MAIN.stLine_BH0IPL.fbLine(stLine:=MAIN.stLine_BH0IPL);
MAIN.stLine_BH0IPL.stStation_BH0IPL01.fbStation(
				stLine:=MAIN.stLine_BH0IPL,
				stStation:=MAIN.stLine_BH0IPL.stStation_BH0IPL01);

END_PROGRAM

// ---- POUs/Program_PIM_Lines/HP/BH0JPL_LineBackground.TcPOU
PROGRAM BH0JPL_LineBackground
VAR
END_VAR

MAIN.stLine_BH0JPL.fbLine(stLine:=MAIN.stLine_BH0JPL);
MAIN.stLine_BH0JPL.stStation_BH0JPL01.fbStation(
				stLine:=MAIN.stLine_BH0JPL,
				stStation:=MAIN.stLine_BH0JPL.stStation_BH0JPL01);

END_PROGRAM

// ---- POUs/Program_PIM_Lines/HP/BH0KPL_LineBackground.TcPOU
PROGRAM BH0KPL_LineBackground
VAR
END_VAR

MAIN.stLine_BH0KPL.fbLine(stLine:=MAIN.stLine_BH0KPL);
MAIN.stLine_BH0KPL.stStation_BH0KPL01.fbStation(
				stLine:=MAIN.stLine_BH0KPL,
				stStation:=MAIN.stLine_BH0KPL.stStation_BH0KPL01);

END_PROGRAM

// ---- POUs/Program_PIM_Lines/HP/BH0LPL_LineBackground.TcPOU
PROGRAM BH0LPL_LineBackground
VAR
END_VAR

MAIN.stLine_BH0LPL.fbLine(stLine:=MAIN.stLine_BH0LPL);
MAIN.stLine_BH0LPL.stStation_BH0LPL01.fbStation(
				stLine:=MAIN.stLine_BH0LPL,
				stStation:=MAIN.stLine_BH0LPL.stStation_BH0LPL01);

END_PROGRAM

// ---- POUs/Program_PIM_Lines/HP/BH0MPL_LineBackground.TcPOU
PROGRAM BH0MPL_LineBackground
VAR
END_VAR

MAIN.stLine_BH0MPL.fbLine(stLine:=MAIN.stLine_BH0MPL);
MAIN.stLine_BH0MPL.stStation_BH0MPL01.fbStation(
				stLine:=MAIN.stLine_BH0MPL,
				stStation:=MAIN.stLine_BH0MPL.stStation_BH0MPL01);

END_PROGRAM

// ---- POUs/Checks/CheckBounds.TcPOU
// Implicitly generated code : DO NOT EDIT
FUNCTION CheckBounds : DINT
VAR_INPUT
	index, lower, upper: DINT;
END_VAR

// Implicitly generated code : Only an Implementation suggestion
{noflow}
IF  index < lower THEN
	GVL_Checks.diCheckBounds := GVL_Checks.diCheckBounds +1;
	CheckBounds := lower;
ELSIF  index > upper THEN
	GVL_Checks.diCheckBounds := GVL_Checks.diCheckBounds +1;
	CheckBounds := upper;
ELSE  
	CheckBounds := index;
END_IF
{flow}

END_FUNCTION

// ---- POUs/Checks/CheckDivDInt.TcPOU
// Implicitly generated code : DO NOT EDIT
FUNCTION CheckDivDInt : DINT
VAR_INPUT
	divisor:DINT;
END_VAR

// Implicitly generated code : Only an Implementation suggestion
{noflow}
IF divisor = 0 THEN
	GVL_Checks.diCheckDivDInt := GVL_Checks.diCheckDivDInt +1;
	CheckDivDInt:=1;
ELSE
	CheckDivDInt:=divisor;
END_IF;
{flow}

END_FUNCTION

// ---- POUs/Checks/CheckDivLInt.TcPOU
// Implicitly generated code : DO NOT EDIT
FUNCTION CheckDivLInt : LINT
VAR_INPUT
	divisor:LINT;
END_VAR

// Implicitly generated code : Only an Implementation suggestion
{noflow}
IF divisor = 0 THEN
GVL_Checks.diCheckDivLInt := GVL_Checks.diCheckDivLInt +1;
	CheckDivLInt:=1;
ELSE
	CheckDivLInt:=divisor;
END_IF;
{flow}

END_FUNCTION

// ---- POUs/Checks/CheckDivLReal.TcPOU
// Implicitly generated code : DO NOT EDIT
FUNCTION CheckDivLReal : LREAL
VAR_INPUT
	divisor:LREAL;
END_VAR

// Implicitly generated code : Only an Implementation suggestion
{noflow}
IF divisor = 0 THEN
	GVL_Checks.diCheckDivLReal := GVL_Checks.diCheckDivLReal +1;
	CheckDivLReal:=1;
ELSE
	CheckDivLReal:=divisor;
END_IF;
{flow}

END_FUNCTION

// ---- POUs/Checks/CheckDivReal.TcPOU
// Implicitly generated code : DO NOT EDIT
FUNCTION CheckDivReal : REAL
VAR_INPUT
	divisor:REAL;
END_VAR

// Implicitly generated code : Only an Implementation suggestion
{noflow}
IF divisor = 0 THEN
GVL_Checks.diCheckDivReal := GVL_Checks.diCheckDivReal +1;
	CheckDivReal:=1;
ELSE
	CheckDivReal:=divisor;
END_IF;
{flow}

END_FUNCTION

// ---- POUs/Checks/CheckLRangeSigned.TcPOU
// Implicitly generated code : DO NOT EDIT
FUNCTION CheckLRangeSigned : LINT
VAR_INPUT
	value, lower, upper: LINT;
END_VAR

// Implicitly generated code : Only an Implementation suggestion
{noflow}
IF (value < lower) THEN
	GVL_Checks.diCheckLRangeSigned := GVL_Checks.diCheckLRangeSigned +1;
	CheckLRangeSigned := lower;
ELSIF(value > upper) THEN
	GVL_Checks.diCheckLRangeSigned := GVL_Checks.diCheckLRangeSigned +1;
	CheckLRangeSigned := upper;
ELSE
	CheckLRangeSigned := value;
END_IF

{flow}

END_FUNCTION

// ---- POUs/Checks/CheckLRangeUnsigned.TcPOU
// Implicitly generated code : DO NOT EDIT
FUNCTION CheckLRangeUnsigned : ULINT
VAR_INPUT
	value, lower, upper: ULINT;
END_VAR

// Implicitly generated code : Only an Implementation suggestion
{noflow}
IF (value < lower) THEN
	GVL_Checks.diCheckLRangeUnsigned := GVL_Checks.diCheckLRangeUnsigned +1;
	CheckLRangeUnsigned := lower;
ELSIF(value > upper) THEN
	GVL_Checks.diCheckLRangeUnsigned := GVL_Checks.diCheckLRangeUnsigned +1;
	CheckLRangeUnsigned := upper;
ELSE
	CheckLRangeUnsigned := value;
END_IF
{flow}

END_FUNCTION

// ---- POUs/Checks/CheckPointer.TcPOU
// Implicitly generated code : DO NOT EDIT
FUNCTION CheckPointer : POINTER TO BYTE
VAR_INPUT 
	ptToTest : POINTER TO BYTE; // Destination address of the pointer
	iSize : DINT;		        // Size of the type the pointer points to. (e.g: 20 for POINTER TO ARRAY [0..9] OF INT) 
	iGran : DINT;		        // Granularity of the pointer access. This is the size of the biggest non-structured data type in the type the pointer points to. (e.g: 2 for POINTER TO ARRAY [0..9] OF INT)
	bWrite: BOOL;		        // Indicates read or write Access. TRUE = write access.
END_VAR

// No standard way of implementation. Fill your own code here
CheckPointer := ptToTest;
IF ptToTest = 0 THEN
	GVL_Checks.diCheckPointer := GVL_Checks.diCheckPointer +1;	
END_IF
{flow}

END_FUNCTION

// ---- POUs/Checks/CheckRangeSigned.TcPOU
// Implicitly generated code : DO NOT EDIT
FUNCTION CheckRangeSigned : DINT
VAR_INPUT
	value, lower, upper: DINT;
END_VAR

// Implicitly generated code : Only an Implementation suggestion
{noflow}
IF (value < lower) THEN
	GVL_Checks.diCheckRangeSigned := GVL_Checks.diCheckRangeSigned +1;
	CheckRangeSigned := lower;
ELSIF(value > upper) THEN
	GVL_Checks.diCheckRangeSigned := GVL_Checks.diCheckRangeSigned +1;
	CheckRangeSigned := upper;
ELSE
	CheckRangeSigned := value;
END_IF
{flow}

END_FUNCTION

// ---- POUs/Checks/CheckRangeUnsigned.TcPOU
// Implicitly generated code : DO NOT EDIT
FUNCTION CheckRangeUnsigned : UDINT
VAR_INPUT
	value, lower, upper: UDINT;
END_VAR

// Implicitly generated code : Only an Implementation suggestion
{noflow}
IF (value < lower) THEN
	GVL_Checks.diCheckRangeUnsigned := GVL_Checks.diCheckRangeUnsigned +1;
	CheckRangeUnsigned := lower;
ELSIF(value > upper) THEN
	GVL_Checks.diCheckRangeUnsigned := GVL_Checks.diCheckRangeUnsigned +1;
	CheckRangeUnsigned := upper;
ELSE
	CheckRangeUnsigned := value;
END_IF
{flow}

END_FUNCTION

// ---- GlobalTextList.TcGTLO
TEXTLIST GlobalTextList
  2028 = '\tWelding plate heaters monitor settings'
  3970 = '\tWelding plate settings'
  1010 = '          Axis brake settings' | pl: 'Ustawienia hamulca'
  2001 = '          Manual mode'
  1107 = '       Actual process data'
  2145 = '       Aux settings'
  810 = '       Axis Calibration'
  1209 = '       Axis specific settings'
  1578 = '       General settings'
  2691 = '       PIM System Active' | pl: '      System PIM aktywny'
  2786 = '      Heat stamp'
  247 = '     %s'
  1851 = '     Heather checking'
  3653 = '    Assembly post station: %s' | pl: 'Stacja montażowa: %s'
  510 = '    Set packing station: %s' | pl: 'Stanowisko pakowania zest.: %s'
  842 = '%.0f'
  641 = '%.1f'
  852 = '%.1f [ % ]'
  5639 = '%.1f [ deg/s ]'
  714 = '%.1f [ mm/s ]'
  2700 = '%.1f [ N ]'
  543 = '%.1f [N]'
  382 = '%.1f [s]'
  978 = '%.2f'
  3732 = '%.2f [ deg ]'
  2622 = '%.2f [ mm ]'
  170 = '%.2f [deg]'
  1131 = '%.3f'
  2649 = '%.3f [ mm ]'
  283 = '%1.2f'
  8 = '%1.f'
  53 = '%2.2f'
  1254 = '%2.f'
  3164 = '%3.f'
  2235 = '%d'
  224 = '%d [deg/s2]'
  2693 = '%d [deg/s]'
  3397 = '%d [deg]'
  4376 = '%f'
  2797 = '%f.2'
  4602 = '%r'
  1 = '%s'
  3861 = "'"
  4535 = '+'
  897 = '+/- %2.2f'
  1682 = '-'
  2248 = '/\\ /\\ /\\      Set NEW    /\\ /\\ /\\' | pl: '/\\ /\\ /\\ Ustaw NOWE /\\ /\\ /\\' | gb: '/\\ /\\ /\\      Set NEW    /\\ /\\ /\\'
  1420 = '1. Adjustment (melting)'
  559 = '1. Choose\nCalibration'
  967 = '2. Connecting parts'
  1292 = '2. Prepare\npart templates'
  33 = '2a- Axis Up \nPart clamp'
  444 = '2b- Axis Dn \nPart clamp'
  2245 = '2c- Close\nWorkCover'
  347 = '3. Evaluate \nresults and exit calib.'
  2022 = '3a- Exit and\nsave result'
  1612 = '3b- Exit \nwithout save'
  393 = '< Act'
  700 = '<A'
  2014 = 'Aby dokonać resetu zaloguj się kartą'
  3442 = 'Aby dokonać resetu zaloguj się:\nswoją kartą'
  4965 = 'Aby dokonać resetu zaloguj się:\nswoją kartą, przykład: id_Pxxxx'
  522 = 'Aby dokonać resetu zaloguj się:\nswoją kartą, przykład: id_Pxxxx\nZalogowane konto ma \nwyświetlać imie i nazwisko'
  610 = 'Aby dokonać resetu zaloguj się:\nswoją kartą, przykład: id_Pxxxx\nZalogowane konto ma wyświetlać imie i nazwisko'
  3960 = 'Acceleration' | pl: 'Przyspieszenie'
  2097 = 'Act axis brake mode'
  2069 = 'Act val. [°C]'
  1347 = 'Activate/deactivate PIM' | pl: 'Włącz/Wyłącz PIM'
  1794 = 'Actual' | pl: 'Aktualne' | gb: 'Actual'
  308 = 'Actual Diference [%]'
  4954 = 'Actual error:' | pl: 'Obecny błąd:'
  1846 = 'Actual position' | pl: 'Obecna pozycja'
  2597 = 'Actual record'
  577 = 'Actual User: %s'
  1769 = 'Actual velocity' | pl: 'Obecna predkosc'
  4416 = 'Actual weight' | pl: 'Obecna waga'
  2569 = 'Actual weight offset [g]'
  1704 = 'Actual weight [g]' | pl: 'Obecna waga [g]'
  2451 = 'Actuator'
  3860 = 'Actuator state'
  685 = 'Adhesion force limit [ N]'
  1373 = 'Adjustment (melting) mode'
  4221 = 'Adjustment distance [mm]'
  2731 = 'Adjustment force [N]'
  743 = 'Adjustment timeout [s]'
  3068 = 'Admin' | pl: 'Administrator'
  1573 = 'Air cut valve acitive' | pl: 'Zawór odcinający powietrze'
  787 = 'Air supply active' | pl: 'Zasilanie pneumatyki włączone'
  1531 = 'Aktualna wartość położenia' | pl: 'Aktualna wartość położenia'
  360 = 'Alarm' | pl: 'Alarm'
  3603 = 'Alarm logging level settings' | pl: 'Poziom logowania alarmów'
  4801 = 'Amount of data exchange'
  4645 = 'Amount of errors'
  3292 = 'Amount of NG commands'
  3000 = 'Amount of OK commands'
  8057 = 'Auto Tare' | pl: 'Auto Tarowanie'
  1112 = 'Available recipe list:' | pl: 'Dostępne receptury:' | gb: 'Avaliable recipes:'
  39 = 'Axis DN WorkStep'
  1058 = 'Axis Down'
  1840 = 'Axis Down WorkStep:'
  561 = 'Axis power control'
  1525 = 'Axis UP WorkStep'
  1687 = 'Axis Up WorkStep:'
  915 = 'Axis Up:'
  195 = 'B02PL production line (LW)' | pl: 'Linia produkcyjna B02PL (LW)'
  1077 = 'BA02PL'
  3259 = 'BA02PL - 1'
  875 = 'BA02PL - 2'
  10432 = 'BA02PL.01.1'
  13845 = 'BA02PL.01.2'
  7111 = 'BA02PL.02'
  17460 = 'BA02PL.03'
  4811 = 'BA02PL.04'
  2952 = 'BA02PL.05'
  12157 = 'BA02PL.06.1'
  3189 = 'BA02PL.06.2'
  1729 = 'BA02PL01_M1'
  223 = 'BA02PL01_M1\nBA02PL01_M2\nBA02PL03'
  2992 = 'BA02PL01_M2'
  5907 = 'BA02PL02'
  2491 = 'BA02PL02\nBA02PL04'
  1317 = 'BA02PL03'
  4279 = 'BA02PL04'
  2606 = 'BA02PL05'
  4490 = 'BA02PL05 - SEQ'
  463 = 'BA02PL06_M1'
  89 = 'BA02PL06_M1\nBA02PL06_M2'
  5291 = 'BA02PL06_M2'
  2816 = 'BA02PL07'
  126 = 'Base pos'
  3252 = 'BB02PL'
  12665 = 'BB02PL.01'
  4132 = 'BB02PL01'
  4062 = 'BH0GPL'
  5405 = 'BH0GPL01_M1'
  4387 = 'BH0GPL01_M2'
  1088 = 'BH0GPL01_M3'
  1316 = 'BH0GPL_M1'
  1606 = 'BH0GPL_M2'
  3567 = 'BH0GPL_M3'
  2067 = 'BH0HPL'
  901 = 'BH0HPL01_M1'
  4474 = 'BH0HPL01_M2'
  1154 = 'BH0HPL01_M3'
  6321 = 'BH0IPL'
  5679 = 'BH0IPL01_M1'
  3354 = 'BH0IPL01_M2'
  197 = 'BH0IPL01_M3'
  6045 = 'BH0JPL'
  1356 = 'BH0JPL01_M1'
  1184 = 'BH0JPL01_M2'
  2515 = 'BH0JPL01_M3'
  3047 = 'BH0KPL'
  4183 = 'BH0KPL01_M1'
  2252 = 'BH0KPL01_M2'
  4613 = 'BH0KPL01_M3'
  778 = 'BH0LPL'
  1170 = 'BH0LPL01_M1'
  5197 = 'BH0LPL01_M2'
  4799 = 'BH0LPL01_M3'
  3559 = 'BH0MPL'
  350 = 'BH0MPL01_M1'
  4743 = 'BH0MPL01_M2'
  316 = 'BH0MPL01_M3'
  2507 = 'Block cardrige'
  3243 = 'Block perform'
  2953 = 'Blocker Down'
  3876 = 'Blocker Entrace'
  3364 = 'Blocker Escape'
  3696 = 'Blocker Input'
  573 = 'Blocker Output'
  3543 = 'Blocker Up'
  1981 = 'BO02PL'
  5711 = 'BO02PL.01'
  14356 = 'BO02PL.02'
  3039 = 'BO02PL01'
  5696 = 'BO02PL02'
  6799 = 'Bottle Detecion From %.2f' | pl: 'Wykrycie Butelki Od %.2f'
  2040 = 'Bottle Detecion To %.2f' | pl: 'Wykrycie Butelki Do %.2f'
  2283 = 'Bottle Incomming'
  3452 = 'Bottle Input'
  8074 = 'Bottle Separation' | pl: 'Oddzielanie Butelek'
  4027 = 'Box target weight: %.3f [kg]' | pl: 'Oczekiwana waga boxa: %.3f [kg]'
  5852 = 'BS02PL'
  8714 = 'BS02PL.01'
  5354 = 'BS02PL01'
  376 = 'BS02PL01_M1'
  701 = 'BS02PL01_M2'
  361 = 'BS02PL03'
  396 = 'BS02PL06_M1'
  649 = 'BS02PL06_M2'
  955 = 'Busy'
  3336 = 'Button On/Off'
  3328 = 'CA03PL'
  1865 = 'CA03PL11'
  2294 = 'CA03PL12'
  2710 = 'CA03PL13'
  514 = 'CA03PL14'
  2017 = 'CA03PL15'
  533 = 'CA03PL16'
  173 = 'CA03PL17'
  3355 = 'CA03PL18'
  200 = 'CA03PL19_M1'
  201 = 'CA03PL19_M2'
  1273 = 'CA03PL20'
  1845 = 'CA03PL21'
  3251 = 'CA03PL22'
  419 = 'Calibration'
  1260 = 'Calibration\nInProgress'
  303 = 'Calibration Target Data'
  179 = 'Camera Contrast'
  437 = 'Camera Exposure Time [us]'
  761 = 'Camera Gain Raw '
  248 = 'Camera Gamma'
  2217 = 'Camera Settings'
  516 = 'Cancel change' | pl: 'Anuluj zmiany' | gb: 'Cancel change'
  2722 = 'Cardrige Chamber'
  557 = 'Cardrige Input'
  90 = 'Cardrige Output'
  4204 = 'Cardrige Table'
  1549 = 'Chamber bussy'
  2795 = 'chamber cardrige'
  2343 = 'Chamber cardrige'
  3054 = 'Chamber work allow'
  7 = 'Check HeatedPlate heaters damage'
  1854 = 'Check heaters'
  109 = 'Check out part dimmenisons tolerance'
  1418 = 'Check part tolerance after contact'
  2132 = 'Check seal'
  5762 = 'Check Vision' | pl: 'Sprawdzanie Wizyjne'
  4753 = 'Check weight' | pl: 'Sprawdzanie wagi'
  5761 = 'Check Weight' | pl: 'Sprawdzanie Wagi'
  3524 = 'Ciśnienie szukania'
  1718 = 'Ciśnienie wprasowania'
  1684 = 'Clean errors' | pl: 'Wyczyść błędy'
  1086 = 'Clear\nStatistic'
  433 = 'Clear History'
  637 = 'CLOSE' | pl: 'ZAMKNIJ'
  1001 = 'Closed'
  508 = 'Closed \n(hiden)'
  654 = 'Closed (hiden)'
  812 = 'CM03PL'
  2300 = 'Cognex settings'
  519 = 'Colision detection EN'
  3451 = 'Colision force treshold'
  2838 = 'Communication Active'
  1552 = 'Communication Cycle Time'
  1968 = 'Communication Cycle Time [s]'
  908 = 'Communication Interval[s]'
  2124 = 'Communication IP'
  520 = 'Communication Ready'
  2647 = 'Confirm change !' | pl: 'Potwierdź zmiany'
  409 = 'Confirm error'
  4955 = 'Confirm PIM Alarm' | pl: 'Potwierdź alarm PIM'
  1985 = 'Confirm PLC Alarm' | pl: 'Potwierdź alarm PLC'
  883 = 'Conn. contact point detec. force [N]'
  785 = 'Connecting distance [mm]'
  285 = 'Connecting force [N]'
  364 = 'Connecting min force to achieve [N]'
  1492 = 'Connecting mode'
  128 = 'Connecting timeout [s]'
  505 = 'Connection Configuration'
  317 = 'Contact point'
  127 = 'Contact point detection force [N]'
  222 = 'Control bag type' | pl: 'Sprawdzaj typ torby'
  3599 = 'Control weight' | pl: 'Sprawdzaj wagę'
  476 = 'Conveyor'
  2212 = 'Conveyor Actuator'
  1708 = 'Convoyer settings'
  596 = 'Cool down time [s]'
  4188 = 'Cooling force first setup [N]'
  1293 = 'Cooling force second setup [N]'
  829 = 'Copmmunicaiton step'
  2215 = 'Copy data TMP -> PLC ?' | pl: 'Przepisać dane TMP -> PLC?'
  213 = 'Copy Recipe Data \nPLC -> TMP ' | pl: 'Kopiuj dane receptury\nPLC -> TMP'
  718 = 'Copy Recipe Data \nTMP -> PLC' | pl: 'Kopiuj dane receptury\nTMP -> PLC'
  235 = 'Cover Cycles: %d'
  187 = 'Cover Cycles: %i'
  3070 = 'CP03PL'
  4182 = 'Current Date Format:'
  1441 = 'Current error code:'
  780 = 'Current error code: %s' | pl: 'Kod aktywnego błędu: %s'
  1847 = 'Current Measure %.0f' | pl: 'Obecny pomiar: %.0f'
  781 = 'Current sensor state:'
  3465 = 'Current:'
  374 = 'Cycle end'
  1106 = 'Cycle time'
  3062 = 'Czas wprasowania'
  1766 = 'DataBase \nError' | pl: 'Błąd\nbazy danych'
  1481 = 'Date format selection by PLC'
  1261 = 'Date format:'
  3466 = 'Deceleration' | pl: 'Zwolnienie'
  461 = 'deg/s'
  80 = 'Delete Selected Recipe' | pl: 'Usuń wybraną recepturę'
  1588 = 'Delete selection ?' | pl: 'Usunąć zaznaczenie ?'
  1649 = 'Description' | pl: 'Opis'
  51 = 'Desired Bag Type:' | pl: 'Oczekiwany typ torby:'
  5000 = 'Details' | pl: 'Szczegoly'
  845 = 'Detection Busy'
  152 = 'Detection Error'
  4153 = 'Detection From: %.0f' | pl: 'Wykrycie Od : %.0f'
  319 = 'Detection Number'
  159 = 'Detection part in fixture EN'
  460 = 'Detection Pass'
  558 = 'Detection Pick'
  1126 = 'Detection To: %.0f' | pl: 'Wykrycie Do: %.0f'
  2408 = 'Detection wait time'
  150 = 'Detection wait time [ms]'
  284 = 'Detection: %d'
  3236 = 'Developer' | pl: 'Programista'
  311 = 'Diagnostics' | pl: 'Diagnostyka'
  790 = 'Diference To Obtain Calib [%]'
  184 = 'Distance between axis'
  3092 = 'DM value: %s' | pl: 'Wartość DM: %s'
  318 = 'Done'
  2821 = 'Doors closed'
  1202 = 'Doors closed NC'
  882 = 'Doors closed NO'
  2864 = 'Dors closed'
  211 = 'Down'
  266 = 'Drawer Unlock\nRequest' | pl: 'Otworz Szuflade'
  4096 = 'dsa'
  3664 = 'dsadasdas'
  782 = 'E-Stop pressed' | pl: 'Wciśnięty E-Stop'
  3564 = 'Edit Types' | pl: 'Edytuj Typy'
  4457 = 'EDIT TYPES' | pl: 'EDYTUJ TYPY'
  1461 = 'Eject perform'
  3847 = 'Eject position'
  6684 = 'EMPTY' | pl: 'OPROZNIANIE'
  4234 = 'Enable' | pl: 'Zezwol'
  667 = 'Enable Auto Tare'
  3962 = 'Enable Cooling force adjustment'
  5457 = 'Enable cooling force adjustment'
  4475 = 'Enable heater burn detection'
  192 = 'Enable heater detection'
  768 = 'Enable logging for:' | pl: 'Włącz logowanie dla:'
  3298 = 'Enable Quick Homing' | pl: 'Wlacz Szybkie Bazowanie'
  1289 = 'Enabled' | pl: 'Zalaczone'
  493 = 'Eng' | pl: 'INZ'
  205 = 'Engineer'
  3485 = 'Entrace cardrige'
  3213 = 'Entrace sensor'
  2333 = 'Error' | pl: 'Błąd'
  1978 = 'Error active' | pl: 'Blad aktywny'
  503 = 'Error Active' | pl: 'Blad Aktywny'
  450 = 'Error Code' | pl: 'Kod błędu'
  2913 = 'Error ID' | pl: 'ID Bledu'
  2502 = 'Error Id: %d' | pl: 'ID Bledu: %d'
  1821 = 'Error Id: %s' | pl: 'ID Bledu: %s'
  747 = 'Error reset' | pl: 'Resetuj Blad'
  4002 = 'Error Reset' | pl: 'Resetuj Blad'
  1083 = 'Error: \n%s' | pl: 'Błąd:\n%s'
  1631 = 'Error: %s' | pl: 'Błąd: %s'
  1670 = 'Errors history' | pl: 'Historia błędow'
  1505 = 'Errors Table' | pl: 'Tablica błędów'
  1037 = 'Escape sensor'
  2477 = 'Exit (no save)' | pl: 'Wyjscie (bez zapisu)'
  494 = 'F'
  1211 = 'Fast movement speed'
  5102 = 'Fast Speed' | pl: 'Predkosc Szybka'
  749 = 'fbStation.fbTimeStats.astTT[INDEX].rStepTime'
  9082 = 'Filling Line'
  1445 = 'Force / Taring'
  1343 = 'Force Filter Time Base [ms]'
  3109 = 'Force Is Stabil'
  563 = 'Force Is Stable'
  2630 = 'Force reference weld \n(part calibration)'
  3752 = 'Force stabil time'
  4609 = 'Force stabil time [ms]'
  1069 = 'Force [ N ]'
  30 = 'General axis parameters'
  1391 = 'General test parameters'
  2615 = 'Green seal'
  265 = 'Hardware error ID'
  6122 = 'Heat Stamp'
  1073 = 'Heat stamp'
  545 = 'Heat stamp\nmake stamp'
  1072 = 'Heat up time [s]'
  31 = 'Heated Plate \nBase Pos'
  1210 = 'Heated Plate \nWork Pos'
  5 = 'Heated plate height'
  1253 = 'Heated plate set temperature [°C]'
  496 = 'Heated plate temp. allowed deviation [°C]'
  4715 = 'Heated plate:'
  4904 = 'Heater current deviation [%]'
  355 = 'Heater current maximal \ndeviation [%]'
  2407 = 'Heater current maximal \ndeviation [A]'
  5670 = 'Heater current maximal deviation [A]'
  2556 = 'Heater current nominal'
  4574 = 'Heater current nominal [A]'
  5131 = 'Heater current readed'
  1364 = 'Heater current readed [A]'
  664 = 'Heaters current \nsensor'
  1218 = 'Heaters Error Active:'
  1212 = 'Heating En'
  710 = 'Heating EN'
  3206 = 'Home Command'
  771 = 'Home Command Perform'
  4702 = 'Home Position' | pl: 'Pozycja bazowa'
  5150 = 'Home position' | pl: 'Pozycja bazowa'
  4942 = 'Homed'
  3737 = 'Homing'
  10691 = 'Hot Plates'
  6738 = 'HotPlate G1\nBH0GPL'
  6341 = 'HotPlate G2\nBH0HPL'
  7041 = 'HotPlate G3\nBH0IPL'
  2165 = 'HotPlate G4\nBH0JPL'
  3188 = 'HotPlate G5\nBH0IPL'
  2228 = 'HotPlate G5\nBH0KPL'
  1110 = 'HotPlate G6\nBH0JPL'
  1511 = 'HotPlate G6\nBH0LPL'
  1183 = 'HotPlate G7\nBH0KPL'
  1259 = 'HotPlate G7\nBH0LPL'
  4503 = 'HotPlate G7\nBH0MPL'
  1061 = 'HotPlates set, station %s'
  13102 = 'HP G1 - BH0GPL'
  10893 = 'HP G2 - BH0HPL'
  3177 = 'HP G3 - BH0IPL'
  16424 = 'HP G4 - BH0JPL'
  12118 = 'HP G5 - BH0KPL'
  6891 = 'HP G6 - BH0LPL'
  6666 = 'HP G7 - BH0MPL'
  1759 = 'I point' | pl: 'Punkt I'
  3407 = 'I: Part presence sensor'
  1570 = 'Identifier | '
  4531 = 'Identifier | IP | Communication Time | Error ID'
  4949 = 'Identifier | IP | Error ID'
  2580 = 'II point' | pl: 'Punkt II'
  611 = 'In Error'
  708 = 'In MOTION'
  2686 = 'In Tare'
  1136 = 'In Valid Position' | pl: 'Poprawna Pozycja'
  630 = 'Info'
  305 = 'Inputs' | pl: 'Wejścia'
  1586 = 'Inputs / Outputs status' | pl: 'Status wejść / wyjść'
  997 = 'IP Adress'
  3121 = 'IP | Identifier | Time | Communication Time | Error ID'
  502 = 'IT (PIM & DB)'
  104 = 'Jog' | pl: 'Jog'
  256 = 'Laser Control'
  168 = 'Last Detection Custom Response'
  2229 = 'Last Detection Data'
  282 = 'Last Detection Number'
  238 = 'Last Detection Parts'
  296 = 'Last Error ID'
  405 = 'Last Home Position' | pl: 'Ostatnia Pozycja Bazowa'
  429 = 'Last Photo Brightness'
  711 = 'Last Photo Contrast'
  100 = 'Last Photo Image Params'
  838 = 'Last Photo Sharpness'
  6137 = 'Last Valid Pos' | pl: 'Ostatnia Poprawna Pozycja'
  2979 = 'Led Blue'
  3795 = 'LED Blue'
  1657 = 'LED Green'
  2225 = 'LED Light Settings'
  246 = 'Led Red'
  3430 = 'LED Red'
  3388 = 'LED Yellow'
  939 = 'LifeBit'
  231 = 'LifeBit Error Time [ms]'
  612 = 'LifeBit machine'
  876 = 'LifeBit PLC'
  162 = 'LifeBit Status'
  2039 = 'Light'
  149 = 'Light Brightness [%]'
  358 = 'Limit exceeded'
  929 = 'Lock'
  1478 = 'Lock part clamp after HP contact'
  1916 = 'Locked'
  3264 = 'Log IN'
  2010 = 'Log out'
  432 = 'Loged User: %s'
  1199 = 'Lower axis'
  775 = 'M1: Iner-Outer Cap'
  68 = 'M2: OuterCap - Mug'
  6 = 'M3: Mug-Bayonet'
  3679 = 'Machine'
  3222 = 'Machine actual state'
  1440 = 'Machine general'
  2524 = 'Machine Indentifier'
  1776 = 'Machine Settings'
  6626 = 'Machine Settings\nBAxxPL'
  1624 = 'Machine Settings\nBSxxPL/BOxxPL\nBBxxPL'
  2885 = 'Machine Settings\nBSxxPL/BOxxPL/\nBBxxPL'
  3761 = 'Machine Settings\nBSxxPL/BOxxPL/BBxxPL'
  2393 = 'Machine Settings\nHotPlate\nBH0xPL'
  3322 = 'Machine Settings\nHP'
  4058 = 'Machine state:'
  116 = 'Machine state: %s'
  881 = 'Machine States'
  2076 = 'Machine WorkStep'
  449 = 'Machine WorkStep:'
  5962 = 'MAIN'
  2492 = 'Main Control' | pl: 'Sekwencja Główna'
  467 = 'Main screen'
  1527 = 'Maintance'
  2531 = 'Maintenance' | pl: 'Utrzymanie Ruchu'
  1994 = 'Make Stamp'
  530 = 'Manual / Service Mode'
  2497 = 'Manual mode' | pl: 'Tryb Reczny'
  2520 = 'MANUAL MODE\nACTIVE' | pl: 'TRYB RECZNY'
  1113 = 'Manual mode \nActive' | pl: 'Tryb reczny'
  1054 = 'Manual mode \nRequest' | pl: 'Tryb reczny'
  2176 = 'MANUAL MODE ACTIVE' | pl: 'TRYB RECZNY AKTYWNY'
  5330 = 'Manual mode active' | pl: 'Tryb reczny aktywny'
  1375 = 'MANUAL MODE REQUEST'
  5383 = 'Manual ON'
  6391 = 'Manual Open' | pl: 'Otworz Recznie'
  398 = 'Marking position'
  3363 = 'Marking time'
  2204 = 'Max motor force (slow)'
  524 = 'Max motor force in slow manual motion'
  5558 = 'Max NOK Bottles %d'
  6104 = 'Max NOK: %d'
  2444 = 'Max powtórzeń detekcji'
  2262 = 'Max. odl. wprasowania'
  946 = 'Maximal position'
  3456 = 'Measure Axis \ndistance'
  3462 = 'Measure HP \nheight'
  2651 = 'Measured' | pl: 'Zmierzone'
  160 = 'Measured Axis distance: %.3f [mm]'
  2196 = 'Measured HP height: %.3f [mm]'
  290 = 'Melting continous force regulation (PI)'
  199 = 'Min. odl. wprasowania'
  776 = 'mm/s'
  1788 = 'Modbus Busy'
  3080 = 'Modbus Error'
  3012 = 'Modbus Error Code'
  919 = 'Modbus TCO - Core statistic'
  2414 = 'Modbus TCP\nCore'
  1772 = 'Modbus TCP - Core statistic'
  1348 = 'Modbus Timeout'
  1529 = 'Monitor OFF time' | pl: 'Monitoruj czas OFF'
  124 = 'Monitor ON time' | pl: 'Monitoruj czas ON'
  1229 = 'Motion error Id: %d' | pl: 'Id Bledu Motion: %d'
  556 = 'Motor acceleration' | pl: 'Przyspieszenie'
  1057 = 'Motor deceleration' | pl: 'Zwolnienie'
  6278 = 'Motor torque limit '
  1650 = 'Motor torque limit [%]'
  2403 = 'Move' | pl: 'Ruch'
  2847 = 'Movement \nInterlock'
  2978 = 'Moving'
  1349 = 'Nb of sets in box: %d [pcs]' | pl: 'L. setów w boxie: %d [szt]'
  4177 = 'Nb of sets on Tray: %d [pcs]' | pl: 'L. setów na palecie: %d [szt]'
  547 = 'New' | pl: 'Nowy'
  1240 = 'New brake mode' | pl: 'Nowy stan hamulca'
  3821 = 'New Tray ' | pl: 'Nowa paleta'
  443 = 'Next step'
  797 = 'NO' | pl: 'NO'
  2754 = 'NOK Bottles Detect %d' | pl: 'Wykrycie Ilosci NOK %d'
  3859 = 'NOK Count: %d' | pl: 'Ilosc NOK: %d'
  112 = 'None' | pl: 'Żaden'
  2261 = 'NO_ONE'
  6097 = 'Offest: %.2f [g]'
  784 = 'Offline work allow'
  4178 = 'ON'
  185 = 'Open'
  2030 = 'Open Entrace Blocker'
  2203 = 'Open Escape Blocker'
  2208 = 'Open WorkCover'
  986 = 'Opened'
  614 = 'Opened (ejected)'
  907 = 'Operator'
  1421 = 'Orange seal'
  1414 = 'Out part dimm. tolerance [mm]'
  1412 = 'Out part set dimmension [mm]'
  1039 = 'Outputs'
  2867 = 'P'
  3359 = 'Parametry procesowe:'
  1976 = 'Part clamp'
  5218 = 'Part load position [mm]'
  1206 = 'Part marking EN'
  410 = 'Part tolerance +/- [mm]'
  3228 = 'Parts done on machine'
  848 = 'Parts NOK: %d'
  103 = 'Parts OK: %d'
  3517 = 'Parts sens'
  108 = 'Perform \nCalibration'
  980 = 'Perform Detection'
  4116 = 'PIM'
  1824 = 'PIM Core Diag.' | pl: 'Rdzen PIM diagnostyka'
  2032 = 'PIM event type: %s' | pl: 'Klasa błędu PIM'
  3242 = 'PIM Last Workstep'
  5946 = 'PIM LifeBit'
  693 = 'PIM States'
  526 = 'PIM system active' | pl: 'Połączenie z PIM aktywne'
  759 = 'PIM work permision'
  1967 = 'PIM work permission' | pl: 'Pozwolenie na pracę z PIM'
  2688 = 'PIM Workstep'
  1188 = 'Place Nr: %d' | pl: 'Gniazdo Nr: %d'
  926 = 'Plate heating EN'
  766 = 'PLC' | pl: 'PLC'
  329 = 'PLC States'
  523 = 'PLC work Permision'
  615 = 'PLC work permission' | pl: 'Pozwolenie na pracę z PLC'
  3751 = 'Port'
  4461 = 'Pos#' | pl: 'Poz#'
  4778 = 'Position Tolerance' | pl: 'Tolerancja Pozycji'
  6643 = 'Position [mm]' | pl: 'Pozycja [mm]'
  4252 = 'Position: %d' | pl: 'Pozycja: %d'
  3373 = 'Positioning Actuator'
  3787 = 'Potwierdz blad %s'
  3297 = 'Power supply ok'
  1546 = 'Power [%]'
  2089 = 'Pozycja wyzwalania'
  5539 = 'Pre Assembly'
  1454 = 'Pre-base position offset [-mm]'
  1473 = 'Pre-connection position offset [-mm]'
  795 = 'Preset Position' | pl: 'Zadana Pozycja'
  3250 = 'Press error: %s'
  1771 = 'Press program step no: %s'
  578 = 'Pressure level do obtain - [kPa]'
  4269 = 'Pressure level [kPa]'
  2301 = 'Program do wybrania'
  2443 = 'Pulls per minute'
  1805 = 'Pulls per second'
  1515 = 'Pump Relay'
  2349 = 'Pump turn on'
  2157 = 'Push position'
  153 = 'Pv'
  1048 = 'Pwr'
  3427 = 'Quality' | pl: 'Jakość'
  5103 = 'Que record'
  2034 = 'Raw' | pl: 'Surowe'
  500 = 'Read Selected Recipe' | pl: 'Odczytaj wybraną recepture'
  599 = 'Ready'
  1046 = 'Ready '
  3431 = 'Received Data'
  1376 = 'Recipe'
  120 = 'Recipe Manager' | pl: 'Menadżer receptur'
  898 = 'Recipe Name: %s' | pl: 'Nazwa receptury: %s'
  1303 = 'Recipes / Test Params'
  1248 = 'Recipes/ test params'
  418 = 'Reference Home Position' | pl: 'Referencyjna Pozycja Bazowa'
  657 = 'Refresh'
  2272 = 'Refresh error:'
  723 = 'Reject \noperation'
  1116 = 'Reload Recipe List' | pl: 'Odśwież listę receptur'
  2436 = 'Repeat Qty' | pl: 'Liczba powtórzeń'
  5803 = 'Request Tare'
  2570 = 'Required OFF time: %.1f [s]'
  2346 = 'Required ON time: %.1f [s]'
  3324 = 'Reset \nCounter'
  48 = 'Reset Counter'
  565 = 'Reset Error' | pl: 'Reset bledu'
  258 = 'Reset error' | pl: 'Reset bledu'
  2437 = 'Reset Marker 1'
  6486 = 'Reset Marker 2'
  447 = 'Reset sequence'
  6841 = 'Reset Tare' | pl: 'Resetuj Tarowanie'
  1156 = 'Reset Transport \nMarker'
  1213 = 'Reset Transport \nMarker 1'
  6345 = 'Reset Transport \nMarker 2'
  4025 = 'Reset Transport Marker'
  1059 = 'Restore' | pl: 'Przywroc'
  721 = 'Restore Last\nValid Pos'
  2692 = 'Rotation Interlock' | pl: 'Zezwolenie Obrotu'
  639 = 'Rotation Request' | pl: 'Rozkaz Obrotu'
  215 = 'RS232 communication' | pl: 'Komunikacja RS232'
  5243 = 'Running Measure: %.2f [g]' | pl: 'Pomiar Ciagly: %.2f [g]'
  957 = 'S01 SealingCork checking EN'
  1186 = 'S19 - EOL'
  4262 = 'S21 - DTL'
  791 = 'Safe HP movement pos [mm]'
  2637 = 'Safety\nRelease'
  1751 = 'Safety diag'
  7230 = 'Safety Door' | pl: 'Drzwi Safety'
  6033 = 'Safety Drawer' | pl: 'Szuflada Safety'
  2796 = 'Safety error' | pl: 'Błąd safety'
  5070 = 'Safety Estop' | pl: 'Estop Safety'
  4264 = 'Safety ok' | pl: 'Safety ok'
  2310 = 'Safety Release' | pl: 'Zezwolenie Safety'
  6247 = 'Save' | pl: 'Zapisz'
  592 = 'Save & Exit' | pl: 'Zapisz & Wyjdz'
  336 = 'Save persistent \ndata' | pl: 'Zapisz dane\nnieulotne'
  742 = 'Save PLC Recipe' | pl: 'Zapisz recepture PLC'
  1080 = 'Save recipe data to file' | pl: 'Zapisz dane receptury do pliku'
  391 = 'Save TMP Recipe' | pl: 'Zapisz recepturę TMP'
  2671 = 'sColumnName_1'
  8132 = 'Seal Color:' | pl: 'Kolor Uszczelki:'
  3435 = 'Send Data'
  2270 = 'Sensor' | pl: 'Sensor'
  6171 = 'Separation ON'
  2509 = 'Separator1 Closing \nDelay [ms]: %d'
  151 = 'Separator1 Closing \nTime[ms]: %d' | pl: 'Czas Zamykania\nSeparatora 1[ms]: %d'
  5707 = 'Separator1 Closing Time[ms]: %d' | pl: 'Czas Zamykania\nSeparatora 1[ms]: %d'
  1308 = 'Serial address'
  3529 = 'Serial communication EN'
  251 = 'Service' | pl: 'Serwis'
  250 = 'SERVICE' | pl: 'SERWIS'
  1220 = 'Service / Manual'
  227 = 'Service possition (lubrication)'
  2406 = 'Servo Details' | pl: 'Servo Szczegoly'
  2328 = 'Set' | pl: 'Ustaw'
  819 = 'Set Intensity'
  3220 = 'Set Offset Position'
  399 = 'Set overview'
  916 = 'Set Power'
  1223 = 'Set val. [°C]'
  734 = 'Set:'
  220 = 'Sets in box: %d [pcs]' | pl: 'Setów w boxie: %d [szt]'
  4160 = 'Sets on tray: %d [pcs]'
  190 = 'Settings' | pl: 'Usrawienia'
  1290 = 'Settings template height'
  813 = 'Signal' | pl: 'Sygnal'
  6057 = 'Single Measure: %.2f [g]' | pl: 'Pojedynczy pomiar :%.2f[g]'
  6112 = 'Single Measurement' | pl: 'Pojedynczy pomiar'
  4699 = 'Slave IP'
  1677 = 'Slow movement speed' | pl: 'Predkosc wolna'
  2604 = 'Slow Speed' | pl: 'Predkosc Wolna'
  2746 = 'Software error ID' | pl: 'ID Bledu'
  899 = 'SonicPress e-stop pressed'
  1247 = 'SonicPress machine:'
  221 = 'SonicPress powered'
  3327 = 'SonicPress work acitve'
  2804 = 'Sonictech welder, station- %s'
  984 = 'Sp'
  2341 = 'Speed setup'
  2753 = 'Speed setup [%]'
  4348 = 'Sprawdzanie odl. końcowej ABS'
  3825 = 'Sprawdzanie odległ. wprasowania DRM'
  3580 = 'Sprawdzanie pozycji wyzwalania'
  5589 = 'Sprawdzenie złożenia SeallingCork'
  4846 = 'Stabil force connecting time [s]'
  2296 = 'Stabilisation Time[ms]: %d' | pl: 'Czas Stabilizacji[ms]: %d'
  6569 = 'Stability Limit: %.2f [%]' | pl: 'Limit Stabilnosci: %.2f[%]'
  2601 = 'Stable' | pl: 'Stabilny'
  4882 = 'Start wait time'
  823 = 'Start wait time [ms]'
  1715 = 'State:' | pl: 'Stan:'
  2231 = 'States'
  1692 = 'States In'
  1161 = 'States Out'
  1833 = 'Station - %s'
  1975 = 'Station data downloaded'
  1632 = 'Station S01-S04'
  4317 = 'Status'
  49 = 'Status / Info'
  123 = 'Step name'
  1728 = 'Step Nr: %d' | pl: 'Nr Kroku: %d'
  4364 = 'Step Number: %d' | pl: 'Numer Kroku: %d'
  125 = 'Step time'
  378 = 'Stop'
  4303 = 'Stop button' | pl: 'Stop'
  5314 = 'Stop Movement' | pl: 'Zatrzymaj'
  306 = 'Stop perform' | pl: 'Zatrzymaj'
  136 = 'S_01'
  2690 = 'S_02'
  880 = 'S_03'
  3461 = 'S_04'
  3935 = 'S_05'
  806 = 'S_06'
  3573 = 'S_07'
  4060 = 'S_08'
  3385 = 'S_09'
  352 = 'S_10'
  1857 = 'S_11'
  965 = 'S_12'
  2452 = 'S_13'
  155 = 'S_14'
  2009 = 'S_15'
  3440 = 'S_16'
  3874 = 'S_17'
  4485 = 'S_18'
  1336 = 'S_19'
  2342 = 'S_20'
  3712 = 'S_21'
  3620 = 'S_22'
  4010 = 'Tare' | pl: 'Tarowanie'
  6877 = 'Tare After Bottles: %d' | pl: 'Tarowanie Po Sztukach: %d'
  5389 = 'Tare Bottle Count: %d' | pl: 'Tarowanie Licznik: %d'
  1087 = 'Tare Offset: %.2f [g]'
  4552 = 'Tare perform' | pl: 'Wykonaj tarowanie'
  2250 = 'Target Brightness'
  554 = 'Target Contrast'
  5176 = 'Target Weight %.2f' | pl: 'Waga docelowa %.2f'
  5468 = 'Target Weight: %d [g]' | pl: 'Waga docelowa: %d[g]'
  453 = 'Taring' | pl: 'Tarowanie'
  1164 = 'Temporary \npermit'
  3318 = 'Temporary permit'
  1207 = 'Tensometer'
  1553 = 'Tensometer Status'
  24 = 'Test mode'
  625 = 'Test mode EN'
  3866 = 'Test perform'
  4433 = 'Test position'
  748 = 'Tests'
  840 = 'Time' | pl: 'Czas'
  3976 = 'Tolerancja poz. wyzwalania'
  952 = 'Total: %d'
  20 = 'Total: %i'
  1979 = 'Touch here and scan Your ID card' | pl: 'Dotknij tutaj i zeskanuj swoją kartę'
  3221 = 'Transfers per minute'
  275 = 'Transfers per second'
  1486 = 'Transporter '
  99 = 'Turn on communication'
  650 = 'Two-hand start input'
  3006 = 'Type in production:' | pl: 'Produkowany typ:'
  5426 = 'Type:' | pl: 'Typ:'
  4716 = 'Type: %s' | pl: 'Typ: %s'
  938 = 'Unit ID'
  480 = 'Unlock'
  673 = 'UP'
  272 = 'Upper axis'
  2634 = 'User loged' | pl: 'Zalogowany'
  1912 = 'User logged' | pl: 'Użytkownik zalogowany'
  167 = 'User login' | pl: 'Login'
  2689 = 'User Name - %s' | pl: 'Nazwa użytk.- %s'
  1800 = 'User Name: %s' | pl: 'Nazwa użytk.: %s'
  91 = 'User Role - %s' | pl: 'Uprawn. użytk.- %s'
  3682 = 'User Role: %s' | pl: 'Updawnienia: %s'
  3042 = 'Ustawienia Kamery:'
  1668 = 'Ustawienia ogolne'
  4202 = 'Uwzględnienie bezpicznej \npozycji dla dwustartu'
  669 = 'Uwzględnienie bezpicznej pozycji dla dwustartu'
  2880 = 'V'
  4019 = 'Vacuum ok'
  686 = 'Vacuum turn on'
  2421 = 'Value' | pl: 'Wartość'
  2419 = 'Valve'
  1957 = 'Valve open'
  1411 = 'Velocity [mm/s]' | pl: 'Predkosc [mm/s]'
  2243 = 'Vision' | pl: 'Wizja'
  1671 = 'VISION' | pl: 'WIZJA'
  143 = 'Vision Max Repeats: %d' | pl: 'Max. Powtorzenia: %d'
  4039 = 'Wait time'
  999 = 'Wait with work'
  3810 = 'Warning'
  1165 = 'Weighing Delay: %d [ms]'
  1850 = 'Weighing Time[ms]: %d' | pl: 'Czas Wazenia[ms]: %d'
  164 = 'Weight'
  5598 = 'WEIGHT' | pl: 'WAZENIE'
  552 = 'Weight settings'
  3680 = 'Weight setup'
  3849 = 'Weight setup [g]'
  839 = 'Weight tolerance' | pl: 'Tolerancja wagi'
  1460 = 'Weight Tolerance %.2f' | pl: 'Tolerancja Wagi %.2f'
  4148 = 'Weight tolerance [g]' | pl: 'Tolerancja wagi [g]'
  2670 = 'Weight tolerance: %.3f [kg]' | pl: 'Tolerancja wagi: %.3f [g]'
  909 = 'Weight Tolerance: %d [g]' | pl: 'Tolerancja wagi : %d [g]'
  827 = 'Weld data:'
  3018 = 'Welding plate settings'
  1230 = 'Work alghorithm:'
  945 = 'Work allow'
  1365 = 'Work Allow'
  3075 = 'Work Command'
  2423 = 'Work Command Perform'
  3400 = 'Work End'
  730 = 'Work in progress'
  1664 = 'Work parameters'
  1475 = 'Wykonanie detekcji '
  1144 = 'X'
  2409 = 'X:'
  964 = 'Y:'
  622 = 'Year - Month'
  621 = 'Year - Week'
  102 = 'YES' | pl: 'TAK'
  770 = '[ mm ]'
  1493 = '[ mm/s ]'
  934 = '[ mm/s² ]'
  567 = '[ N ]'
  572 = '[ s ]'
  389 = '[ s ] '
  5794 = '[% ]'
  3909 = '[bar]'
  3506 = '[deg]'
  3091 = '[mm]'
  5768 = '[°C ]'
  1883 = '^^ Set NEW ^^' | pl: '^^ Ustaw NOWE ^^'
  1045 = '^^^ Confirm change !!! ^^^' | pl: '^^^ Potwierdź zmianę !!! ^^^'
END_TEXTLIST

// ---- VISUs/New Visus/HomeVisuBA02PL.TcVIS
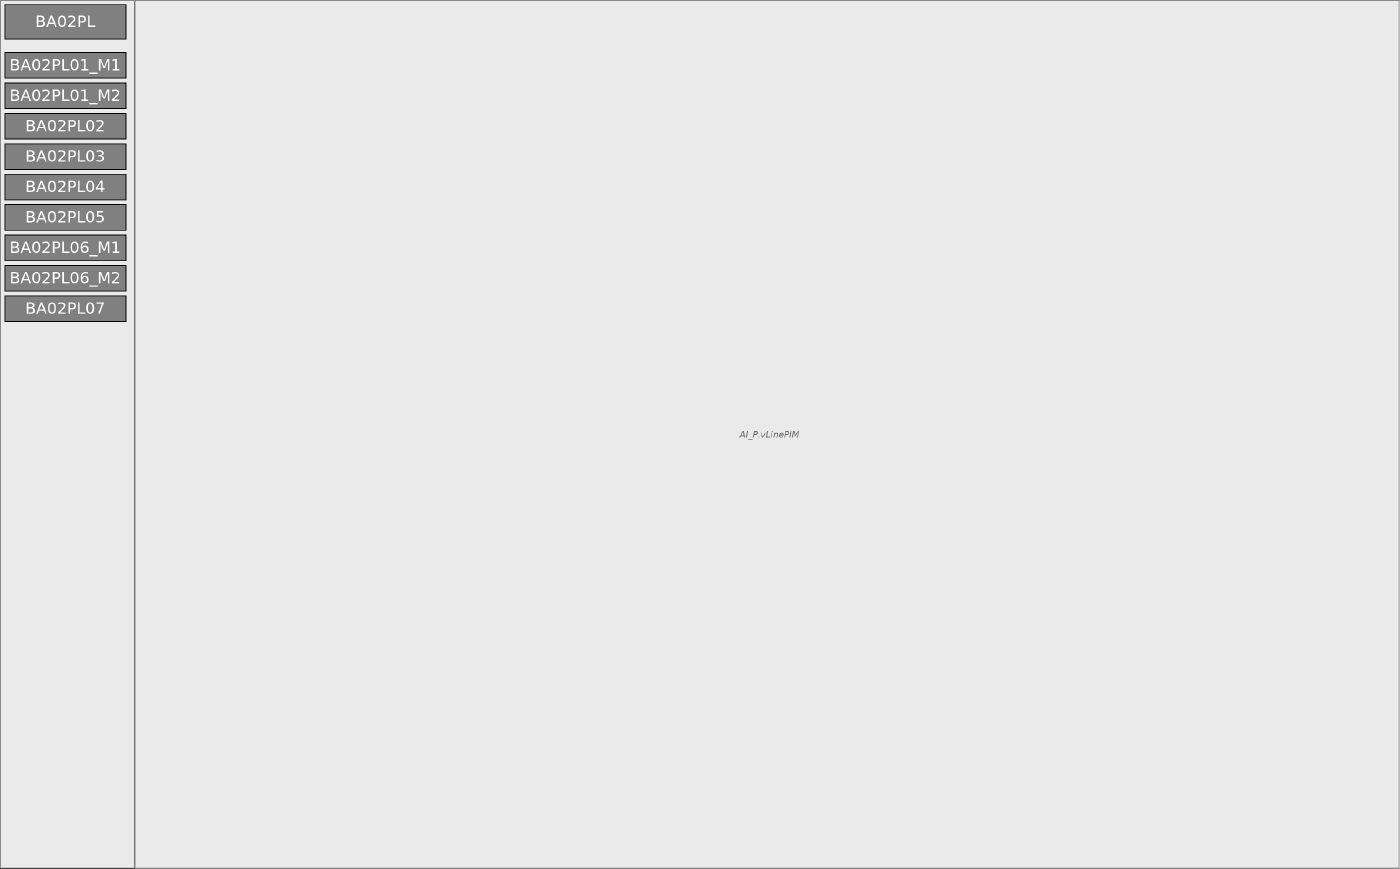
VISUALIZATION HomeVisuBA02PL  // 1610x1000
    Rectangle (0,0 155x1000)
    Frame (155,0 1460x1000)
        shows AI_P.vLinePIM(fbPIM := MAIN.stLine_BA02PL.fbLine)
        shows AI_P.vStationPIM(fbPIM := MAIN.fb_Filler_A_Machine.fbPIM)
        shows AI_P.vStationPIM(fbPIM := MAIN.fb_Cork_Machine.fbPIM)
        shows AI_P.vStationPIM(fbPIM := MAIN.fb_1_SonicTech_SonictechUSW.fbPIM)
        shows AI_P.vStationPIM(fbPIM := MAIN.fb_Filler_B_Machine.fbPIM)
        shows AI_P.vStationPIM(fbPIM := MAIN.fb_2_SonicTech_SonictechUSW.fbPIM)
        shows AI_P.vStationPIM(fbPIM := MAIN.fb_UnderPressure_Tester_Machine.fbPIM)
        shows AI_P.vStationPIM(fbPIM := MAIN.fb_Sticker_Machine.fbPIM)
        shows AI_P.vStationPIM(fbPIM := MAIN.fb_Laser_Machine.fbPIM)
        shows AI_P.vStationPIM(fbPIM := MAIN.fbWeighingTunel.fbTableControl.fbPIM)
        shows AircomLibrary.vStationPIM(fbPIM := MAIN.fbS19_2_EOL3.fbPIM)
        shows AircomLibrary.vStationPIM(fbPIM := MAIN.fbS20_AssemblyPost.fbPIM)
        shows AircomLibrary.vStationPIM(fbPIM := MAIN.fbS21_DetectionTunel.fbPIM)
        shows AircomLibrary.vStationPIM(fbPIM := MAIN.fbS22_SetPackingStation.fbPIM)
        p2766960713: GVL.fbSqlCore
        p2683556743: GVL.stLJ20_DTL_WorkParams
        p3043078949: MAIN.fbLL19_1_EOL3
        p1709583229: GVL.stLL19_EOL_Settings_I
        p2719655782: MAIN.fbLL19_2_EOL3
        p3094409976: GVL.stLL19_EOL_Settings_II
        p74549115: 'Left chamber'
        p3369830373: 'Right chamber'
        p3445515547: MAIN.fbLS06
        p3589162504: GVL_IO.stLS01_HoseCutter
        p458721708: MAIN.fbLS01_HoseCutter
        p3390713232: MAIN.fbLS04_1_Station
        p1393785898: MAIN.fbLS04_2_Station
        p3419948967: MAIN.fbLS05_1_Station
        p1389434397: MAIN.fbLS05_2_Station
        p422258626: MAIN.fbLS04_1_Crimper
        p417943029: MAIN.fbLS05_1_Crimper
        p2149742200: MAIN.fbLS04_2_Crimper
        p2178948175: MAIN.fbLS05_2_Crimper
        p180551898: MAIN.fbS03
        p2110009420: MAIN.fbLS02_InsertAssy
        p2404496545: MAIN.fbLS02_Station
        p4166419511: MAIN.fbLS03_Station
        p1449093633: MAIN.fbLS06_V2
        p898092448: GVL.Hose_Tester_Params_V2
        p589997586: GVL.Hose_Tester_Params_V2.iPickedHose
        p1762866656: MAIN.fbS03
        p504628598: MAIN.fbLS02_InsertAssy
        p1957019379: MAIN.fbLS06_V2
        p1712759876: GVL.Hose_Tester_Params_V2
        p3689475492: GVL.Hose_Tester_Params_V2.iPickedHose
        p1628323955: MAIN.fbS21_DetectionTunel.fbPIM
        p2913222893: MAIN.fbS22_SetPackingStation.fbPIM
    Rectangle (5,5 140x40), "BA02PL"
        OnMouseDown: FrameSelectionChange Selection=SelectedFrame=cd818c81-a6c5-4ab8-9515-1ee8055884ac, GlobSel=AssignType=Directly, SelType=Locally
    Rectangle (5,60 140x30), "BA02PL01_M1"
        OnMouseDown: FrameSelectionChange Selection=SelectedFrame=cd818c81-a6c5-4ab8-9515-1ee8055884ac, Selection=1, GlobSel=AssignType=Directly, SelType=Locally
    Rectangle (5,165 140x30), "BA02PL03"
        OnMouseDown: FrameSelectionChange Selection=SelectedFrame=cd818c81-a6c5-4ab8-9515-1ee8055884ac, Selection=4, GlobSel=AssignType=Directly, SelType=Locally
    Rectangle (5,95 140x30), "BA02PL01_M2"
        OnMouseDown: FrameSelectionChange Selection=SelectedFrame=cd818c81-a6c5-4ab8-9515-1ee8055884ac, Selection=2, GlobSel=AssignType=Directly, SelType=Locally
    Rectangle (5,130 140x30), "BA02PL02"
        OnMouseDown: FrameSelectionChange Selection=SelectedFrame=cd818c81-a6c5-4ab8-9515-1ee8055884ac, Selection=3, GlobSel=AssignType=Directly, SelType=Locally
    Rectangle (5,200 140x30), "BA02PL04"
        OnMouseDown: FrameSelectionChange Selection=SelectedFrame=cd818c81-a6c5-4ab8-9515-1ee8055884ac, Selection=5, GlobSel=AssignType=Directly, SelType=Locally
    Rectangle (5,235 140x30), "BA02PL05"
        OnMouseDown: FrameSelectionChange Selection=SelectedFrame=cd818c81-a6c5-4ab8-9515-1ee8055884ac, Selection=6, GlobSel=AssignType=Directly, SelType=Locally
    Rectangle (5,305 140x30), "BA02PL06_M2"
        OnMouseDown: FrameSelectionChange Selection=SelectedFrame=cd818c81-a6c5-4ab8-9515-1ee8055884ac, Selection=8, GlobSel=AssignType=Directly, SelType=Locally
    Rectangle (5,270 140x30), "BA02PL06_M1"
        OnMouseDown: FrameSelectionChange Selection=SelectedFrame=cd818c81-a6c5-4ab8-9515-1ee8055884ac, Selection=7, GlobSel=AssignType=Directly, SelType=Locally
    Rectangle (5,340 140x30), "BA02PL07"
        OnMouseDown: FrameSelectionChange Selection=SelectedFrame=cd818c81-a6c5-4ab8-9515-1ee8055884ac, Selection=9, GlobSel=AssignType=Directly, SelType=Locally
END_VISUALIZATION

// ---- VISUs/New Visus/HomeVisuBB02PL.TcVIS
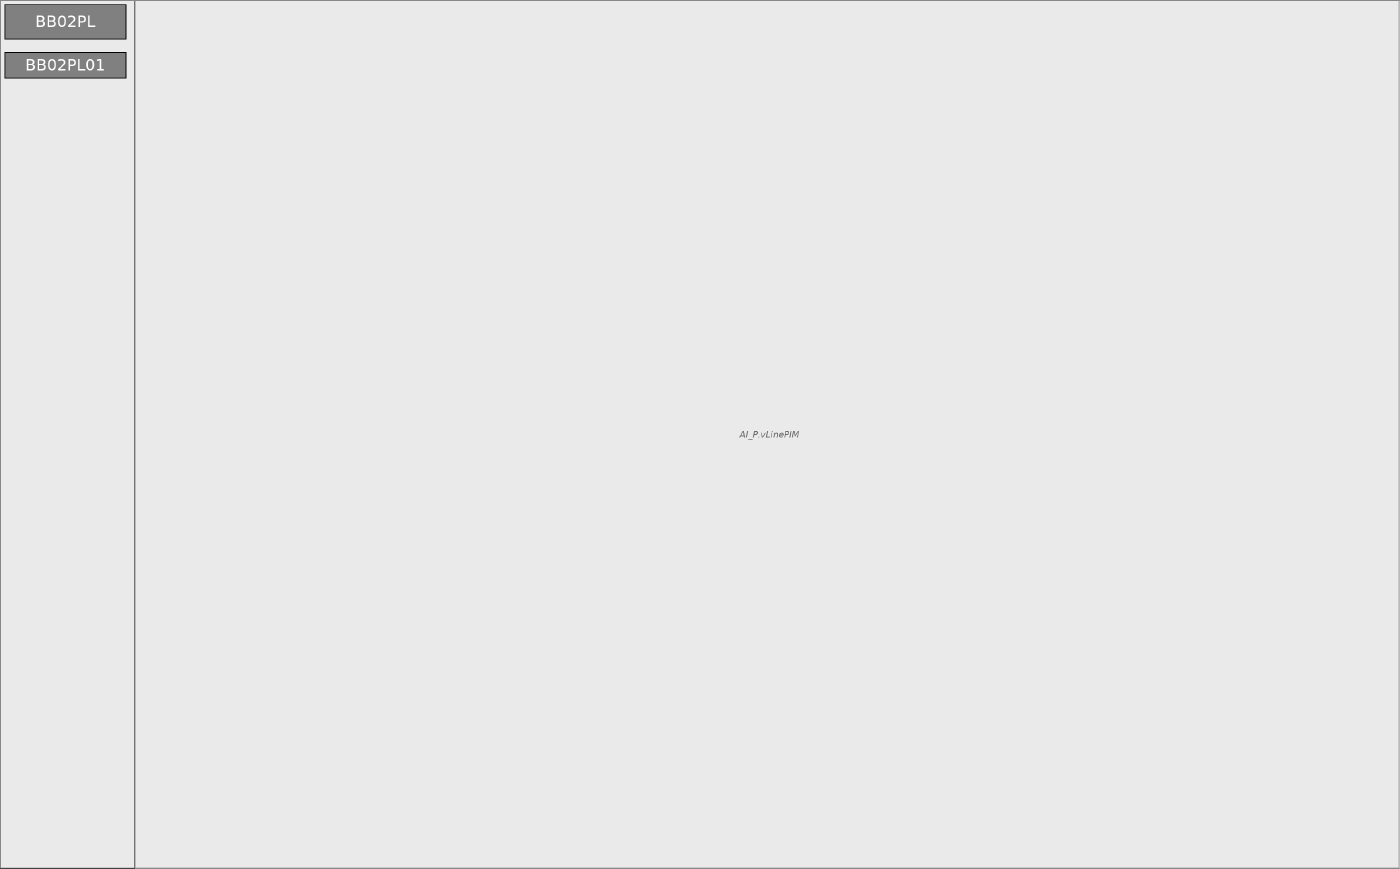
VISUALIZATION HomeVisuBB02PL  // 1610x1000
    Rectangle (0,0 155x1000)
    Frame (155,0 1460x1000)
        shows AI_P.vLinePIM(fbPIM := MAIN.stLine_BB02PL.fbLine)
        shows AI_P.vStationPIM(fbPIM := MAIN.fbS02_BearingPress.fbPIM)
        shows AircomLibrary.vStationPIM(fbPIM := MAIN.fbS13_FrontFan.fbPIM)
        shows AircomLibrary.vStationPIM(fbPIM := MAIN.fbS14_AssemblyPost.fbPIM)
        shows AircomLibrary.vStationPIM(fbPIM := MAIN.fbS12_Hios.fbPIM)
        shows AircomLibrary.vStationPIM(fbPIM := MAIN.fbS15_AssemblyPost.fbPIM)
        shows AircomLibrary.vStationPIM(fbPIM := MAIN.fbS16_SonictechUSW.fbPIM)
        shows AircomLibrary.vStationPIM(fbPIM := MAIN.fbS17_SonictechUSW.fbPIM)
        shows AircomLibrary.vStationPIM(fbPIM := MAIN.fbS19_1_EOL3.fbPIM)
        shows AircomLibrary.vStationPIM(fbPIM := MAIN.fbS19_2_EOL3.fbPIM)
        shows AircomLibrary.vStationPIM(fbPIM := MAIN.fbS20_AssemblyPost.fbPIM)
        shows AircomLibrary.vStationPIM(fbPIM := MAIN.fbS21_DetectionTunel.fbPIM)
        shows AircomLibrary.vStationPIM(fbPIM := MAIN.fbS22_SetPackingStation.fbPIM)
        shows AircomLibrary.vStationPIM()
        p2766960713: GVL.fbSqlCore
        p2683556743: GVL.stLJ20_DTL_WorkParams
        p3043078949: MAIN.fbLL19_1_EOL3
        p1709583229: GVL.stLL19_EOL_Settings_I
        p2719655782: MAIN.fbLL19_2_EOL3
        p3094409976: GVL.stLL19_EOL_Settings_II
        p74549115: 'Left chamber'
        p3369830373: 'Right chamber'
        p3445515547: MAIN.fbLS06
        p3589162504: GVL_IO.stLS01_HoseCutter
        p458721708: MAIN.fbLS01_HoseCutter
        p3390713232: MAIN.fbLS04_1_Station
        p1393785898: MAIN.fbLS04_2_Station
        p3419948967: MAIN.fbLS05_1_Station
        p1389434397: MAIN.fbLS05_2_Station
        p422258626: MAIN.fbLS04_1_Crimper
        p417943029: MAIN.fbLS05_1_Crimper
        p2149742200: MAIN.fbLS04_2_Crimper
        p2178948175: MAIN.fbLS05_2_Crimper
        p180551898: MAIN.fbS03
        p2110009420: MAIN.fbLS02_InsertAssy
        p2404496545: MAIN.fbLS02_Station
        p4166419511: MAIN.fbLS03_Station
        p1449093633: MAIN.fbLS06_V2
        p898092448: GVL.Hose_Tester_Params_V2
        p589997586: GVL.Hose_Tester_Params_V2.iPickedHose
        p1762866656: MAIN.fbS03
        p504628598: MAIN.fbLS02_InsertAssy
        p1957019379: MAIN.fbLS06_V2
        p1712759876: GVL.Hose_Tester_Params_V2
        p3689475492: GVL.Hose_Tester_Params_V2.iPickedHose
        p1628323955: MAIN.fbS21_DetectionTunel.fbPIM
        p2913222893: MAIN.fbS22_SetPackingStation.fbPIM
    Rectangle (5,5 140x40), "BB02PL"
        OnMouseDown: FrameSelectionChange Selection=SelectedFrame=cd818c81-a6c5-4ab8-9515-1ee8055884ac, GlobSel=AssignType=Directly, SelType=Locally
    Rectangle (5,60 140x30), "BB02PL01"
        OnMouseDown: FrameSelectionChange Selection=SelectedFrame=cd818c81-a6c5-4ab8-9515-1ee8055884ac, Selection=1, GlobSel=AssignType=Directly, SelType=Locally
END_VISUALIZATION

// ---- VISUs/New Visus/HomeVisuBH0GPL.TcVIS
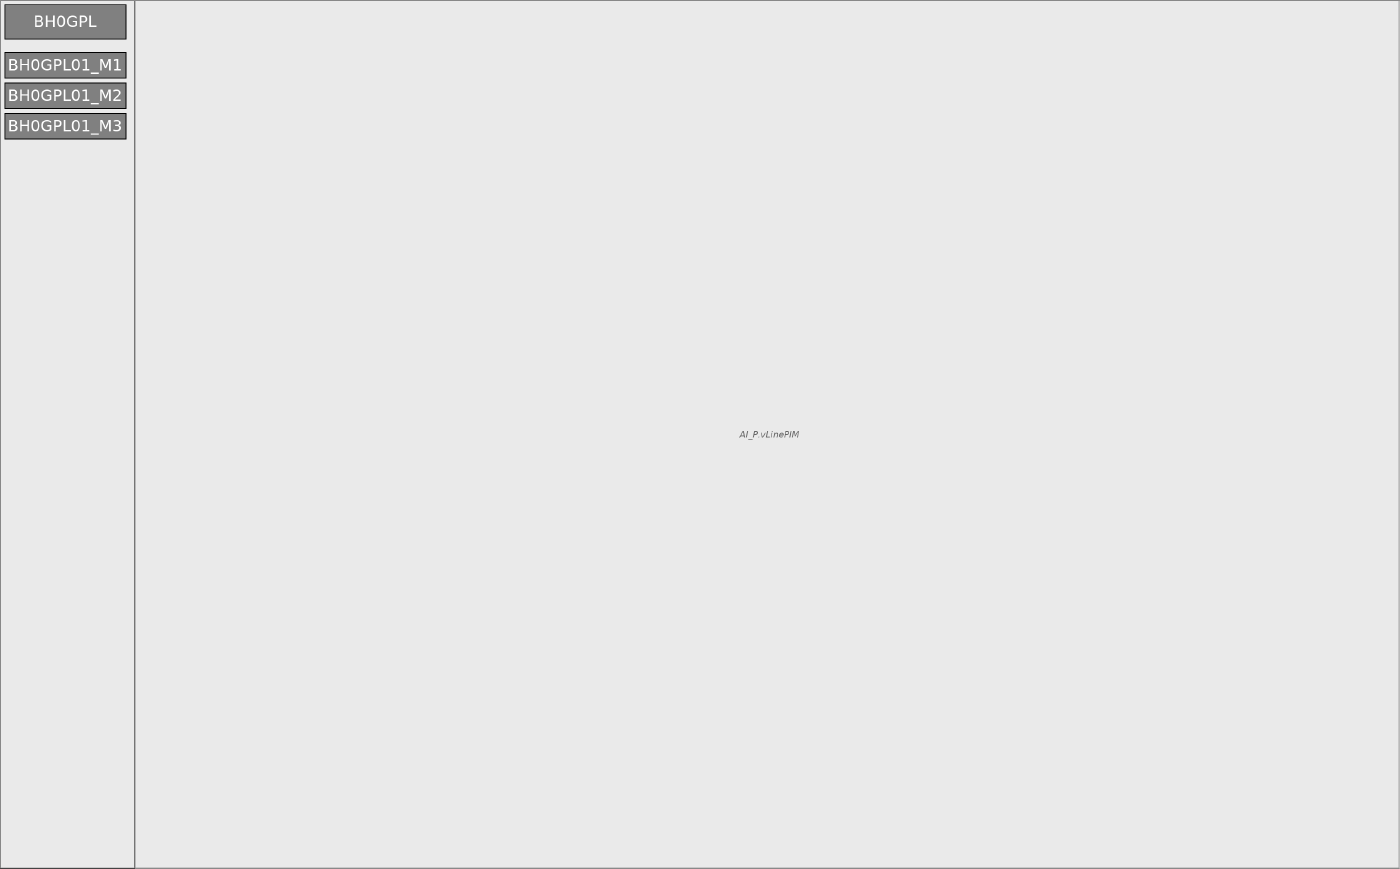
VISUALIZATION HomeVisuBH0GPL  // 1610x1000
    Rectangle (0,0 155x1000)
    Frame (155,0 1460x1000)
        shows AI_P.vLinePIM(fbPIM := MAIN.stLine_BH0GPL.fbLine)
        shows AI_P.vStationPIM(fbPIM := MAIN.fbHotPlate_G1_M1.fbPIM)
        shows AI_P.vStationPIM(fbPIM := MAIN.fbHotPlate_G1_M2.fbPIM)
        shows AI_P.vStationPIM(fbPIM := MAIN.fbHotPlate_G1_M3.fbPIM)
        shows AircomLibrary.vStationPIM(fbPIM := MAIN.fbS14_AssemblyPost.fbPIM)
        shows AircomLibrary.vStationPIM(fbPIM := MAIN.fbS15_AssemblyPost.fbPIM)
        shows AircomLibrary.vStationPIM(fbPIM := MAIN.fbS16_SonictechUSW.fbPIM)
        shows AircomLibrary.vStationPIM(fbPIM := MAIN.fbS17_SonictechUSW.fbPIM)
        shows AircomLibrary.vStationPIM(fbPIM := MAIN.fbS19_1_EOL3.fbPIM)
        shows AircomLibrary.vStationPIM(fbPIM := MAIN.fbS19_2_EOL3.fbPIM)
        shows AircomLibrary.vStationPIM(fbPIM := MAIN.fbS20_AssemblyPost.fbPIM)
        shows AircomLibrary.vStationPIM(fbPIM := MAIN.fbS21_DetectionTunel.fbPIM)
        shows AircomLibrary.vStationPIM(fbPIM := MAIN.fbS22_SetPackingStation.fbPIM)
        shows AircomLibrary.vStationPIM()
        p2766960713: GVL.fbSqlCore
        p2683556743: GVL.stLJ20_DTL_WorkParams
        p3043078949: MAIN.fbLL19_1_EOL3
        p1709583229: GVL.stLL19_EOL_Settings_I
        p2719655782: MAIN.fbLL19_2_EOL3
        p3094409976: GVL.stLL19_EOL_Settings_II
        p74549115: 'Left chamber'
        p3369830373: 'Right chamber'
        p3445515547: MAIN.fbLS06
        p3589162504: GVL_IO.stLS01_HoseCutter
        p458721708: MAIN.fbLS01_HoseCutter
        p3390713232: MAIN.fbLS04_1_Station
        p1393785898: MAIN.fbLS04_2_Station
        p3419948967: MAIN.fbLS05_1_Station
        p1389434397: MAIN.fbLS05_2_Station
        p422258626: MAIN.fbLS04_1_Crimper
        p417943029: MAIN.fbLS05_1_Crimper
        p2149742200: MAIN.fbLS04_2_Crimper
        p2178948175: MAIN.fbLS05_2_Crimper
        p180551898: MAIN.fbS03
        p2110009420: MAIN.fbLS02_InsertAssy
        p2404496545: MAIN.fbLS02_Station
        p4166419511: MAIN.fbLS03_Station
        p1449093633: MAIN.fbLS06_V2
        p898092448: GVL.Hose_Tester_Params_V2
        p589997586: GVL.Hose_Tester_Params_V2.iPickedHose
        p1762866656: MAIN.fbS03
        p504628598: MAIN.fbLS02_InsertAssy
        p1957019379: MAIN.fbLS06_V2
        p1712759876: GVL.Hose_Tester_Params_V2
        p3689475492: GVL.Hose_Tester_Params_V2.iPickedHose
        p1628323955: MAIN.fbS21_DetectionTunel.fbPIM
        p2913222893: MAIN.fbS22_SetPackingStation.fbPIM
    Rectangle (5,5 140x40), "BH0GPL"
        OnMouseDown: FrameSelectionChange Selection=SelectedFrame=cd818c81-a6c5-4ab8-9515-1ee8055884ac, GlobSel=AssignType=Directly, SelType=Locally
    Rectangle (5,60 140x30), "BH0GPL01_M1"
        OnMouseDown: FrameSelectionChange Selection=SelectedFrame=cd818c81-a6c5-4ab8-9515-1ee8055884ac, Selection=1, GlobSel=AssignType=Directly, SelType=Locally
    Rectangle (5,95 140x30), "BH0GPL01_M2"
        OnMouseDown: FrameSelectionChange Selection=SelectedFrame=cd818c81-a6c5-4ab8-9515-1ee8055884ac, Selection=2, GlobSel=AssignType=Directly, SelType=Locally
    Rectangle (5,130 140x30), "BH0GPL01_M3"
        OnMouseDown: FrameSelectionChange Selection=SelectedFrame=cd818c81-a6c5-4ab8-9515-1ee8055884ac, Selection=3, GlobSel=AssignType=Directly, SelType=Locally
END_VISUALIZATION

// ---- VISUs/New Visus/HomeVisuBH0HPL.TcVIS
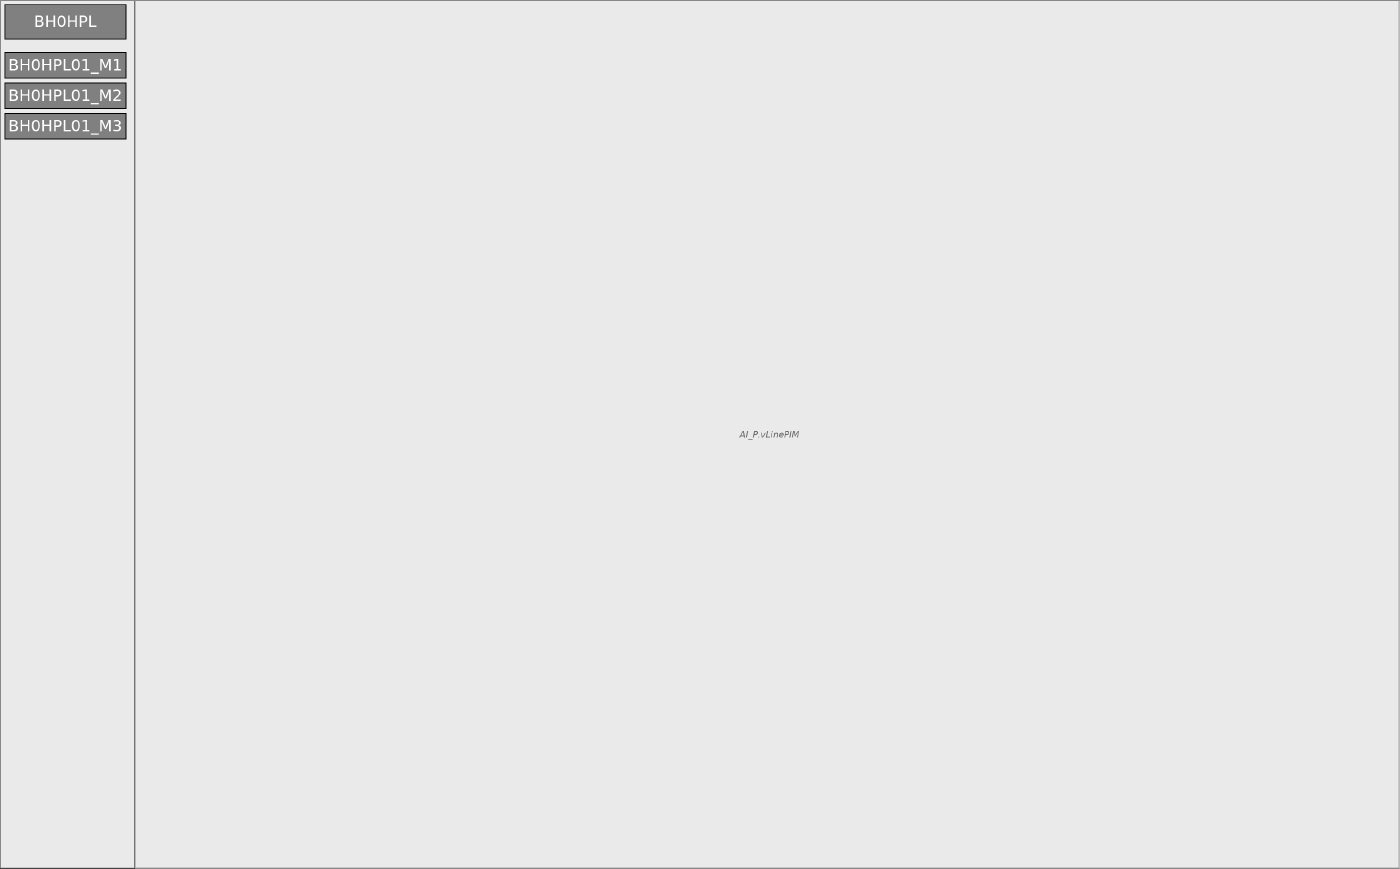
VISUALIZATION HomeVisuBH0HPL  // 1610x1000
    Rectangle (0,0 155x1000)
    Frame (155,0 1460x1000)
        shows AI_P.vLinePIM(fbPIM := MAIN.stLine_BH0HPL.fbLine)
        shows AI_P.vStationPIM(fbPIM := MAIN.fbHotPlate_G2_M1.fbPIM)
        shows AI_P.vStationPIM(fbPIM := MAIN.fbHotPlate_G2_M2.fbPIM)
        shows AI_P.vStationPIM(fbPIM := MAIN.fbHotPlate_G2_M3.fbPIM)
        shows AircomLibrary.vStationPIM(fbPIM := MAIN.fbS14_AssemblyPost.fbPIM)
        shows AircomLibrary.vStationPIM(fbPIM := MAIN.fbS15_AssemblyPost.fbPIM)
        shows AircomLibrary.vStationPIM(fbPIM := MAIN.fbS16_SonictechUSW.fbPIM)
        shows AircomLibrary.vStationPIM(fbPIM := MAIN.fbS17_SonictechUSW.fbPIM)
        shows AircomLibrary.vStationPIM(fbPIM := MAIN.fbS19_1_EOL3.fbPIM)
        shows AircomLibrary.vStationPIM(fbPIM := MAIN.fbS19_2_EOL3.fbPIM)
        shows AircomLibrary.vStationPIM(fbPIM := MAIN.fbS20_AssemblyPost.fbPIM)
        shows AircomLibrary.vStationPIM(fbPIM := MAIN.fbS21_DetectionTunel.fbPIM)
        shows AircomLibrary.vStationPIM(fbPIM := MAIN.fbS22_SetPackingStation.fbPIM)
        shows AircomLibrary.vStationPIM()
        p2766960713: GVL.fbSqlCore
        p2683556743: GVL.stLJ20_DTL_WorkParams
        p3043078949: MAIN.fbLL19_1_EOL3
        p1709583229: GVL.stLL19_EOL_Settings_I
        p2719655782: MAIN.fbLL19_2_EOL3
        p3094409976: GVL.stLL19_EOL_Settings_II
        p74549115: 'Left chamber'
        p3369830373: 'Right chamber'
        p3445515547: MAIN.fbLS06
        p3589162504: GVL_IO.stLS01_HoseCutter
        p458721708: MAIN.fbLS01_HoseCutter
        p3390713232: MAIN.fbLS04_1_Station
        p1393785898: MAIN.fbLS04_2_Station
        p3419948967: MAIN.fbLS05_1_Station
        p1389434397: MAIN.fbLS05_2_Station
        p422258626: MAIN.fbLS04_1_Crimper
        p417943029: MAIN.fbLS05_1_Crimper
        p2149742200: MAIN.fbLS04_2_Crimper
        p2178948175: MAIN.fbLS05_2_Crimper
        p180551898: MAIN.fbS03
        p2110009420: MAIN.fbLS02_InsertAssy
        p2404496545: MAIN.fbLS02_Station
        p4166419511: MAIN.fbLS03_Station
        p1449093633: MAIN.fbLS06_V2
        p898092448: GVL.Hose_Tester_Params_V2
        p589997586: GVL.Hose_Tester_Params_V2.iPickedHose
        p1762866656: MAIN.fbS03
        p504628598: MAIN.fbLS02_InsertAssy
        p1957019379: MAIN.fbLS06_V2
        p1712759876: GVL.Hose_Tester_Params_V2
        p3689475492: GVL.Hose_Tester_Params_V2.iPickedHose
        p1628323955: MAIN.fbS21_DetectionTunel.fbPIM
        p2913222893: MAIN.fbS22_SetPackingStation.fbPIM
    Rectangle (5,5 140x40), "BH0HPL"
        OnMouseDown: FrameSelectionChange Selection=SelectedFrame=cd818c81-a6c5-4ab8-9515-1ee8055884ac, GlobSel=AssignType=Directly, SelType=Locally
    Rectangle (5,60 140x30), "BH0HPL01_M1"
        OnMouseDown: FrameSelectionChange Selection=SelectedFrame=cd818c81-a6c5-4ab8-9515-1ee8055884ac, Selection=1, GlobSel=AssignType=Directly, SelType=Locally
    Rectangle (5,95 140x30), "BH0HPL01_M2"
        OnMouseDown: FrameSelectionChange Selection=SelectedFrame=cd818c81-a6c5-4ab8-9515-1ee8055884ac, Selection=2, GlobSel=AssignType=Directly, SelType=Locally
    Rectangle (5,130 140x30), "BH0HPL01_M3"
        OnMouseDown: FrameSelectionChange Selection=SelectedFrame=cd818c81-a6c5-4ab8-9515-1ee8055884ac, Selection=3, GlobSel=AssignType=Directly, SelType=Locally
END_VISUALIZATION

// ---- VISUs/New Visus/HomeVisuBH0IPL.TcVIS
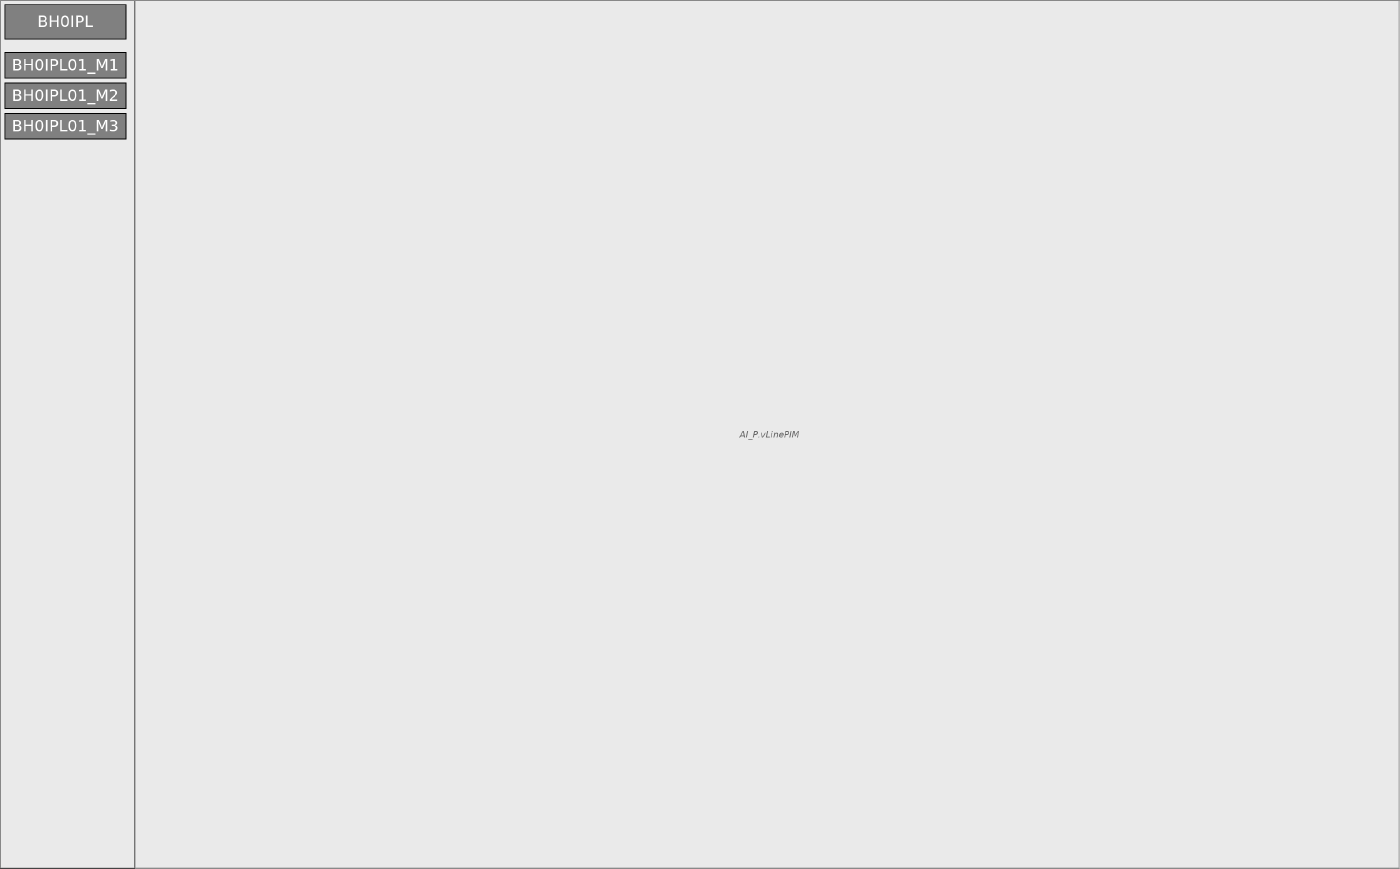
VISUALIZATION HomeVisuBH0IPL  // 1610x1000
    Rectangle (0,0 155x1000)
    Frame (155,0 1460x1000)
        shows AI_P.vLinePIM(fbPIM := MAIN.stLine_BH0IPL.fbLine)
        shows AI_P.vStationPIM(fbPIM := MAIN.fbHotPlate_G3_M1.fbPIM)
        shows AI_P.vStationPIM(fbPIM := MAIN.fbHotPlate_G3_M2.fbPIM)
        shows AI_P.vStationPIM(fbPIM := MAIN.fbHotPlate_G3_M3.fbPIM)
        shows AircomLibrary.vStationPIM(fbPIM := MAIN.fbS14_AssemblyPost.fbPIM)
        shows AircomLibrary.vStationPIM(fbPIM := MAIN.fbS15_AssemblyPost.fbPIM)
        shows AircomLibrary.vStationPIM(fbPIM := MAIN.fbS16_SonictechUSW.fbPIM)
        shows AircomLibrary.vStationPIM(fbPIM := MAIN.fbS17_SonictechUSW.fbPIM)
        shows AircomLibrary.vStationPIM(fbPIM := MAIN.fbS19_1_EOL3.fbPIM)
        shows AircomLibrary.vStationPIM(fbPIM := MAIN.fbS19_2_EOL3.fbPIM)
        shows AircomLibrary.vStationPIM(fbPIM := MAIN.fbS20_AssemblyPost.fbPIM)
        shows AircomLibrary.vStationPIM(fbPIM := MAIN.fbS21_DetectionTunel.fbPIM)
        shows AircomLibrary.vStationPIM(fbPIM := MAIN.fbS22_SetPackingStation.fbPIM)
        shows AircomLibrary.vStationPIM()
        p2766960713: GVL.fbSqlCore
        p2683556743: GVL.stLJ20_DTL_WorkParams
        p3043078949: MAIN.fbLL19_1_EOL3
        p1709583229: GVL.stLL19_EOL_Settings_I
        p2719655782: MAIN.fbLL19_2_EOL3
        p3094409976: GVL.stLL19_EOL_Settings_II
        p74549115: 'Left chamber'
        p3369830373: 'Right chamber'
        p3445515547: MAIN.fbLS06
        p3589162504: GVL_IO.stLS01_HoseCutter
        p458721708: MAIN.fbLS01_HoseCutter
        p3390713232: MAIN.fbLS04_1_Station
        p1393785898: MAIN.fbLS04_2_Station
        p3419948967: MAIN.fbLS05_1_Station
        p1389434397: MAIN.fbLS05_2_Station
        p422258626: MAIN.fbLS04_1_Crimper
        p417943029: MAIN.fbLS05_1_Crimper
        p2149742200: MAIN.fbLS04_2_Crimper
        p2178948175: MAIN.fbLS05_2_Crimper
        p180551898: MAIN.fbS03
        p2110009420: MAIN.fbLS02_InsertAssy
        p2404496545: MAIN.fbLS02_Station
        p4166419511: MAIN.fbLS03_Station
        p1449093633: MAIN.fbLS06_V2
        p898092448: GVL.Hose_Tester_Params_V2
        p589997586: GVL.Hose_Tester_Params_V2.iPickedHose
        p1762866656: MAIN.fbS03
        p504628598: MAIN.fbLS02_InsertAssy
        p1957019379: MAIN.fbLS06_V2
        p1712759876: GVL.Hose_Tester_Params_V2
        p3689475492: GVL.Hose_Tester_Params_V2.iPickedHose
        p1628323955: MAIN.fbS21_DetectionTunel.fbPIM
        p2913222893: MAIN.fbS22_SetPackingStation.fbPIM
    Rectangle (5,5 140x40), "BH0IPL"
        OnMouseDown: FrameSelectionChange Selection=SelectedFrame=cd818c81-a6c5-4ab8-9515-1ee8055884ac, GlobSel=AssignType=Directly, SelType=Locally
    Rectangle (5,60 140x30), "BH0IPL01_M1"
        OnMouseDown: FrameSelectionChange Selection=SelectedFrame=cd818c81-a6c5-4ab8-9515-1ee8055884ac, Selection=1, GlobSel=AssignType=Directly, SelType=Locally
    Rectangle (5,95 140x30), "BH0IPL01_M2"
        OnMouseDown: FrameSelectionChange Selection=SelectedFrame=cd818c81-a6c5-4ab8-9515-1ee8055884ac, Selection=2, GlobSel=AssignType=Directly, SelType=Locally
    Rectangle (5,130 140x30), "BH0IPL01_M3"
        OnMouseDown: FrameSelectionChange Selection=SelectedFrame=cd818c81-a6c5-4ab8-9515-1ee8055884ac, Selection=3, GlobSel=AssignType=Directly, SelType=Locally
END_VISUALIZATION

// ---- VISUs/New Visus/HomeVisuBH0JPL.TcVIS
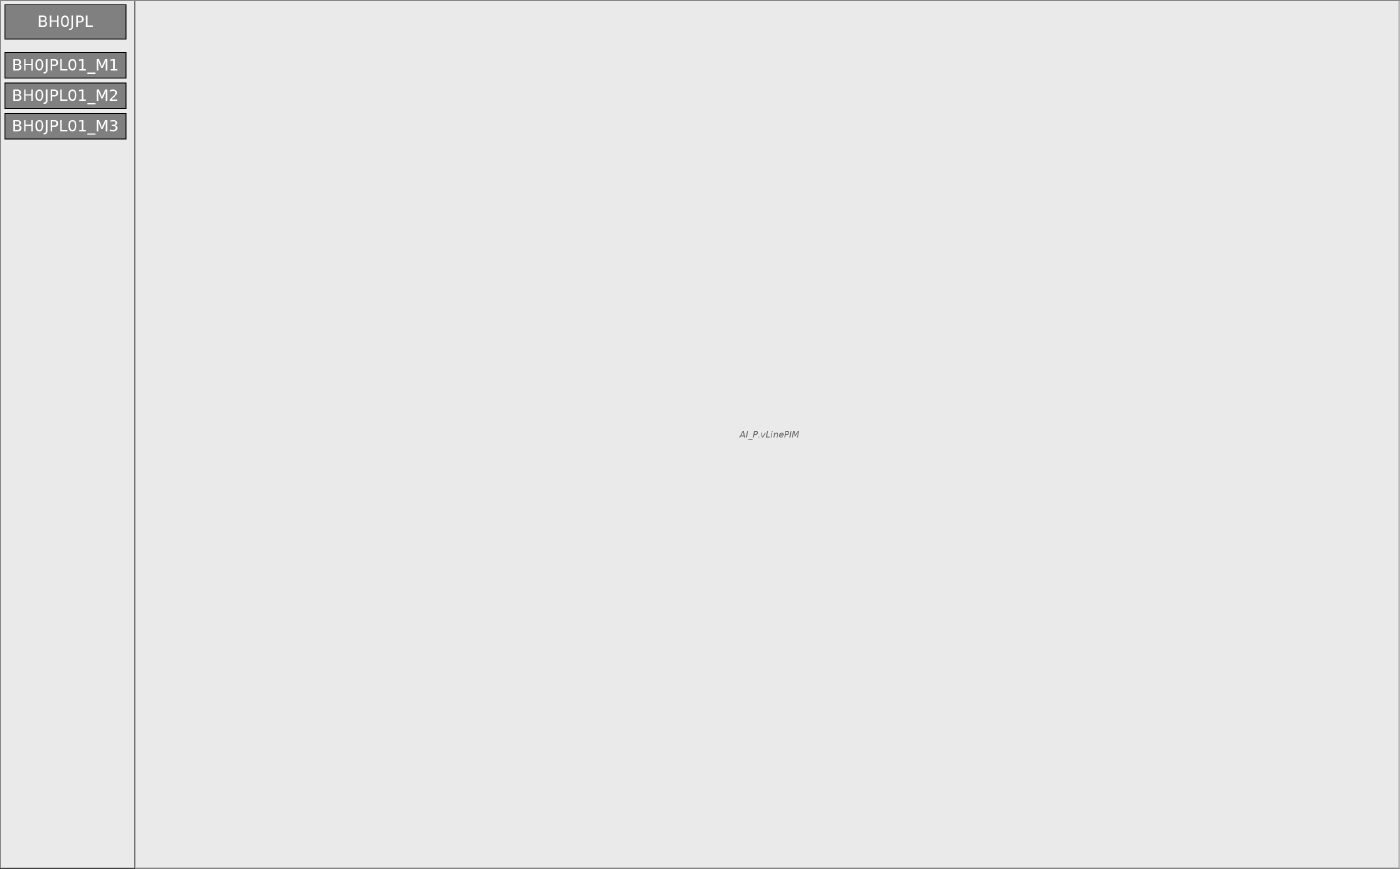
VISUALIZATION HomeVisuBH0JPL  // 1610x1000
    Rectangle (0,0 155x1000)
    Frame (155,0 1460x1000)
        shows AI_P.vLinePIM(fbPIM := MAIN.stLine_BH0JPL.fbLine)
        shows AI_P.vStationPIM(fbPIM := MAIN.fbHotPlate_G4_M1.fbPIM)
        shows AI_P.vStationPIM(fbPIM := MAIN.fbHotPlate_G4_M2.fbPIM)
        shows AI_P.vStationPIM(fbPIM := MAIN.fbHotPlate_G4_M3.fbPIM)
        shows AircomLibrary.vStationPIM(fbPIM := MAIN.fbS14_AssemblyPost.fbPIM)
        shows AircomLibrary.vStationPIM(fbPIM := MAIN.fbS15_AssemblyPost.fbPIM)
        shows AircomLibrary.vStationPIM(fbPIM := MAIN.fbS16_SonictechUSW.fbPIM)
        shows AircomLibrary.vStationPIM(fbPIM := MAIN.fbS17_SonictechUSW.fbPIM)
        shows AircomLibrary.vStationPIM(fbPIM := MAIN.fbS19_1_EOL3.fbPIM)
        shows AircomLibrary.vStationPIM(fbPIM := MAIN.fbS19_2_EOL3.fbPIM)
        shows AircomLibrary.vStationPIM(fbPIM := MAIN.fbS20_AssemblyPost.fbPIM)
        shows AircomLibrary.vStationPIM(fbPIM := MAIN.fbS21_DetectionTunel.fbPIM)
        shows AircomLibrary.vStationPIM(fbPIM := MAIN.fbS22_SetPackingStation.fbPIM)
        shows AircomLibrary.vStationPIM()
        p2766960713: GVL.fbSqlCore
        p2683556743: GVL.stLJ20_DTL_WorkParams
        p3043078949: MAIN.fbLL19_1_EOL3
        p1709583229: GVL.stLL19_EOL_Settings_I
        p2719655782: MAIN.fbLL19_2_EOL3
        p3094409976: GVL.stLL19_EOL_Settings_II
        p74549115: 'Left chamber'
        p3369830373: 'Right chamber'
        p3445515547: MAIN.fbLS06
        p3589162504: GVL_IO.stLS01_HoseCutter
        p458721708: MAIN.fbLS01_HoseCutter
        p3390713232: MAIN.fbLS04_1_Station
        p1393785898: MAIN.fbLS04_2_Station
        p3419948967: MAIN.fbLS05_1_Station
        p1389434397: MAIN.fbLS05_2_Station
        p422258626: MAIN.fbLS04_1_Crimper
        p417943029: MAIN.fbLS05_1_Crimper
        p2149742200: MAIN.fbLS04_2_Crimper
        p2178948175: MAIN.fbLS05_2_Crimper
        p180551898: MAIN.fbS03
        p2110009420: MAIN.fbLS02_InsertAssy
        p2404496545: MAIN.fbLS02_Station
        p4166419511: MAIN.fbLS03_Station
        p1449093633: MAIN.fbLS06_V2
        p898092448: GVL.Hose_Tester_Params_V2
        p589997586: GVL.Hose_Tester_Params_V2.iPickedHose
        p1762866656: MAIN.fbS03
        p504628598: MAIN.fbLS02_InsertAssy
        p1957019379: MAIN.fbLS06_V2
        p1712759876: GVL.Hose_Tester_Params_V2
        p3689475492: GVL.Hose_Tester_Params_V2.iPickedHose
        p1628323955: MAIN.fbS21_DetectionTunel.fbPIM
        p2913222893: MAIN.fbS22_SetPackingStation.fbPIM
    Rectangle (5,5 140x40), "BH0JPL"
        OnMouseDown: FrameSelectionChange Selection=SelectedFrame=cd818c81-a6c5-4ab8-9515-1ee8055884ac, GlobSel=AssignType=Directly, SelType=Locally
    Rectangle (5,60 140x30), "BH0JPL01_M1"
        OnMouseDown: FrameSelectionChange Selection=SelectedFrame=cd818c81-a6c5-4ab8-9515-1ee8055884ac, Selection=1, GlobSel=AssignType=Directly, SelType=Locally
    Rectangle (5,95 140x30), "BH0JPL01_M2"
        OnMouseDown: FrameSelectionChange Selection=SelectedFrame=cd818c81-a6c5-4ab8-9515-1ee8055884ac, Selection=2, GlobSel=AssignType=Directly, SelType=Locally
    Rectangle (5,130 140x30), "BH0JPL01_M3"
        OnMouseDown: FrameSelectionChange Selection=SelectedFrame=cd818c81-a6c5-4ab8-9515-1ee8055884ac, Selection=3, GlobSel=AssignType=Directly, SelType=Locally
END_VISUALIZATION

// ---- VISUs/New Visus/HomeVisuBH0KPL.TcVIS
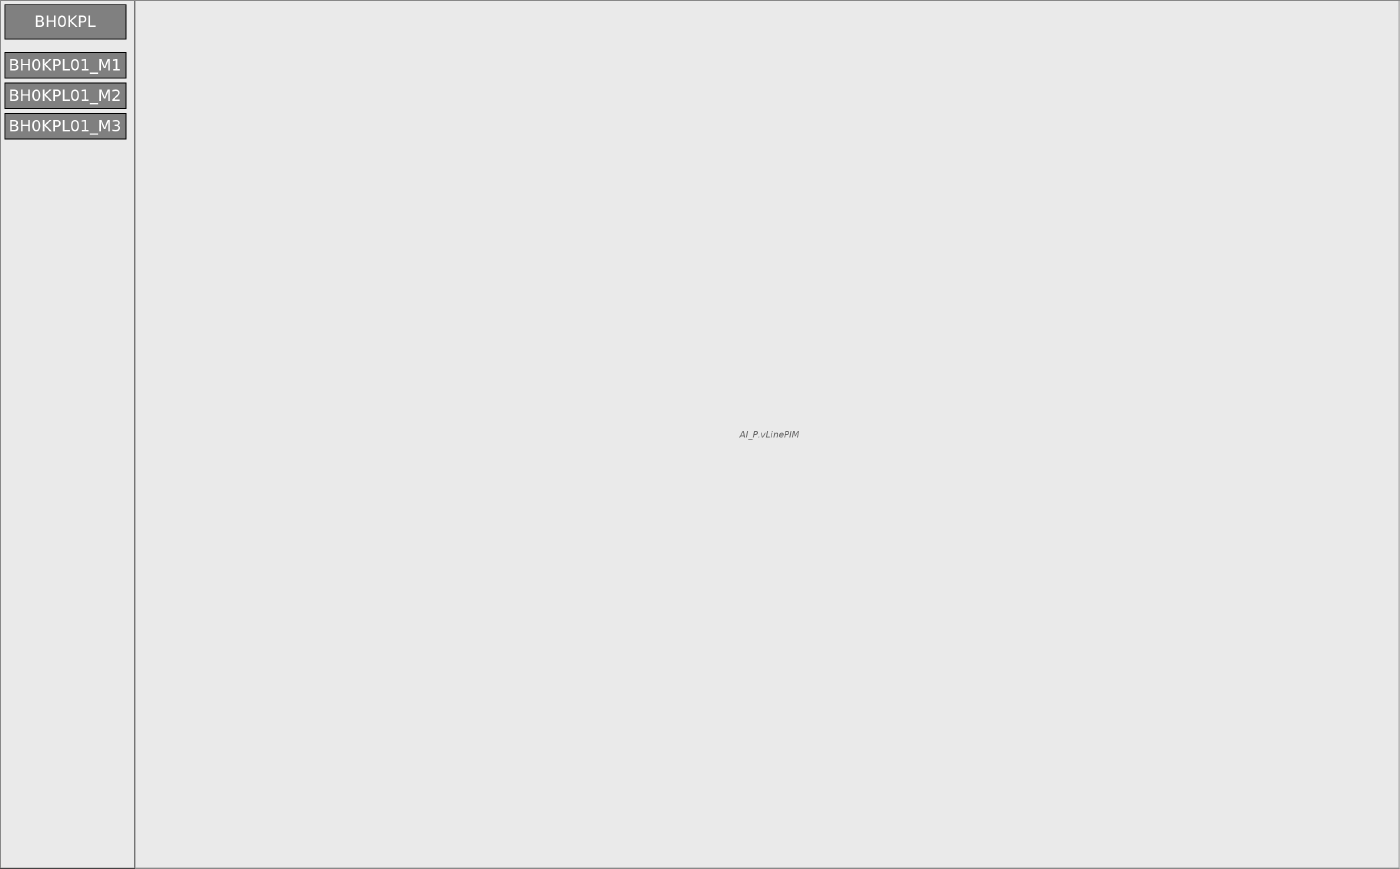
VISUALIZATION HomeVisuBH0KPL  // 1610x1000
    Rectangle (0,0 155x1000)
    Frame (155,0 1460x1000)
        shows AI_P.vLinePIM(fbPIM := MAIN.stLine_BH0KPL.fbLine)
        shows AI_P.vStationPIM(fbPIM := MAIN.fbHotPlate_G5_M1.fbPIM)
        shows AI_P.vStationPIM(fbPIM := MAIN.fbHotPlate_G5_M2.fbPIM)
        shows AI_P.vStationPIM(fbPIM := MAIN.fbHotPlate_G5_M3.fbPIM)
        shows AircomLibrary.vStationPIM(fbPIM := MAIN.fbS14_AssemblyPost.fbPIM)
        shows AircomLibrary.vStationPIM(fbPIM := MAIN.fbS15_AssemblyPost.fbPIM)
        shows AircomLibrary.vStationPIM(fbPIM := MAIN.fbS16_SonictechUSW.fbPIM)
        shows AircomLibrary.vStationPIM(fbPIM := MAIN.fbS17_SonictechUSW.fbPIM)
        shows AircomLibrary.vStationPIM(fbPIM := MAIN.fbS19_1_EOL3.fbPIM)
        shows AircomLibrary.vStationPIM(fbPIM := MAIN.fbS19_2_EOL3.fbPIM)
        shows AircomLibrary.vStationPIM(fbPIM := MAIN.fbS20_AssemblyPost.fbPIM)
        shows AircomLibrary.vStationPIM(fbPIM := MAIN.fbS21_DetectionTunel.fbPIM)
        shows AircomLibrary.vStationPIM(fbPIM := MAIN.fbS22_SetPackingStation.fbPIM)
        shows AircomLibrary.vStationPIM()
        p2766960713: GVL.fbSqlCore
        p2683556743: GVL.stLJ20_DTL_WorkParams
        p3043078949: MAIN.fbLL19_1_EOL3
        p1709583229: GVL.stLL19_EOL_Settings_I
        p2719655782: MAIN.fbLL19_2_EOL3
        p3094409976: GVL.stLL19_EOL_Settings_II
        p74549115: 'Left chamber'
        p3369830373: 'Right chamber'
        p3445515547: MAIN.fbLS06
        p3589162504: GVL_IO.stLS01_HoseCutter
        p458721708: MAIN.fbLS01_HoseCutter
        p3390713232: MAIN.fbLS04_1_Station
        p1393785898: MAIN.fbLS04_2_Station
        p3419948967: MAIN.fbLS05_1_Station
        p1389434397: MAIN.fbLS05_2_Station
        p422258626: MAIN.fbLS04_1_Crimper
        p417943029: MAIN.fbLS05_1_Crimper
        p2149742200: MAIN.fbLS04_2_Crimper
        p2178948175: MAIN.fbLS05_2_Crimper
        p180551898: MAIN.fbS03
        p2110009420: MAIN.fbLS02_InsertAssy
        p2404496545: MAIN.fbLS02_Station
        p4166419511: MAIN.fbLS03_Station
        p1449093633: MAIN.fbLS06_V2
        p898092448: GVL.Hose_Tester_Params_V2
        p589997586: GVL.Hose_Tester_Params_V2.iPickedHose
        p1762866656: MAIN.fbS03
        p504628598: MAIN.fbLS02_InsertAssy
        p1957019379: MAIN.fbLS06_V2
        p1712759876: GVL.Hose_Tester_Params_V2
        p3689475492: GVL.Hose_Tester_Params_V2.iPickedHose
        p1628323955: MAIN.fbS21_DetectionTunel.fbPIM
        p2913222893: MAIN.fbS22_SetPackingStation.fbPIM
    Rectangle (5,5 140x40), "BH0KPL"
        OnMouseDown: FrameSelectionChange Selection=SelectedFrame=cd818c81-a6c5-4ab8-9515-1ee8055884ac, GlobSel=AssignType=Directly, SelType=Locally
    Rectangle (5,60 140x30), "BH0KPL01_M1"
        OnMouseDown: FrameSelectionChange Selection=SelectedFrame=cd818c81-a6c5-4ab8-9515-1ee8055884ac, Selection=1, GlobSel=AssignType=Directly, SelType=Locally
    Rectangle (5,95 140x30), "BH0KPL01_M2"
        OnMouseDown: FrameSelectionChange Selection=SelectedFrame=cd818c81-a6c5-4ab8-9515-1ee8055884ac, Selection=2, GlobSel=AssignType=Directly, SelType=Locally
    Rectangle (5,130 140x30), "BH0KPL01_M3"
        OnMouseDown: FrameSelectionChange Selection=SelectedFrame=cd818c81-a6c5-4ab8-9515-1ee8055884ac, Selection=3, GlobSel=AssignType=Directly, SelType=Locally
END_VISUALIZATION

// ---- VISUs/New Visus/HomeVisuBH0LPL.TcVIS
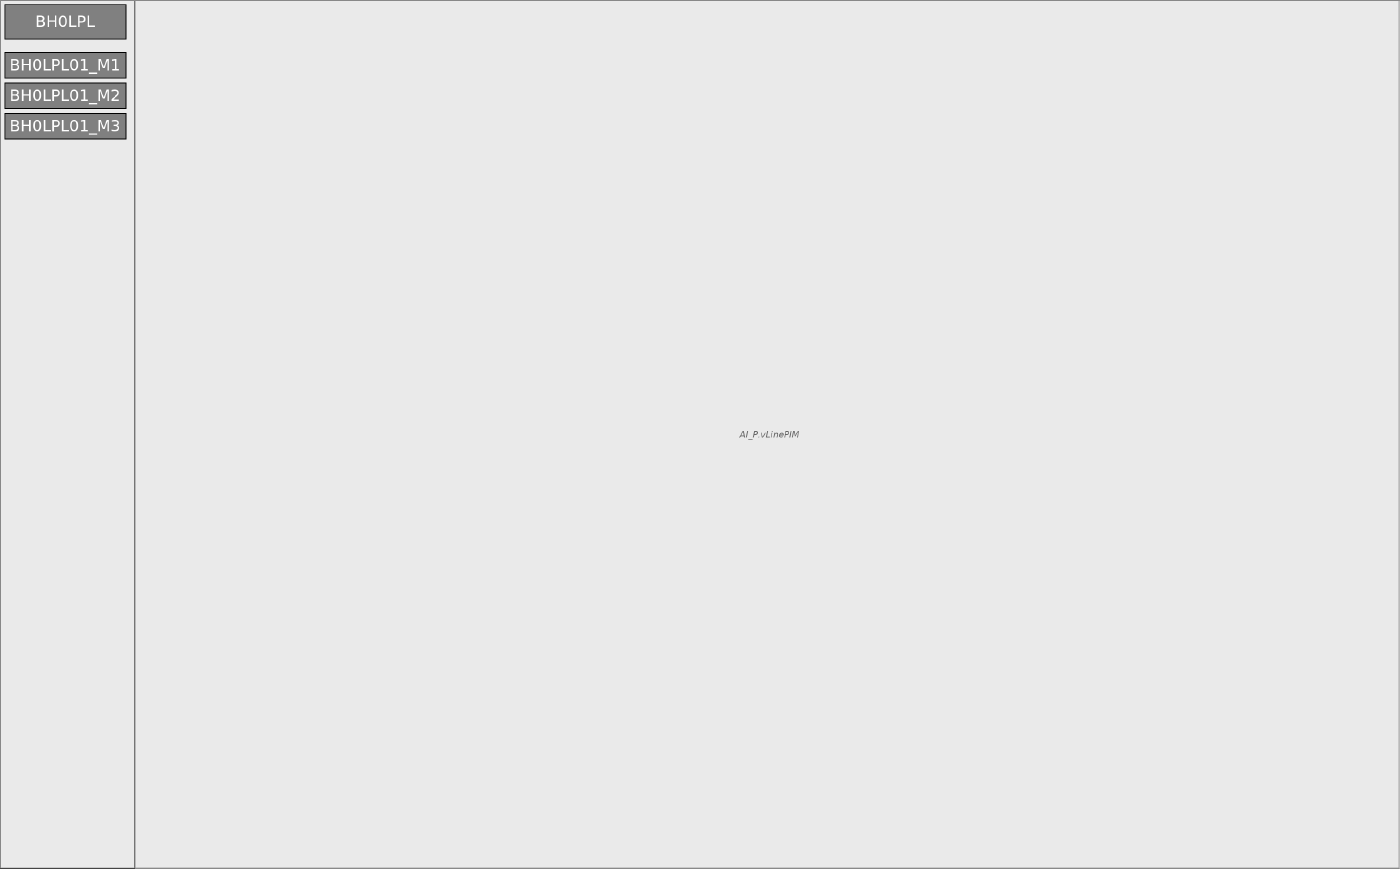
VISUALIZATION HomeVisuBH0LPL  // 1610x1000
    Rectangle (0,0 155x1000)
    Frame (155,0 1460x1000)
        shows AI_P.vLinePIM(fbPIM := MAIN.stLine_BH0LPL.fbLine)
        shows AI_P.vStationPIM(fbPIM := MAIN.fbHotPlate_G6_M1.fbPIM)
        shows AI_P.vStationPIM(fbPIM := MAIN.fbHotPlate_G6_M2.fbPIM)
        shows AI_P.vStationPIM(fbPIM := MAIN.fbHotPlate_G6_M3.fbPIM)
        shows AircomLibrary.vStationPIM(fbPIM := MAIN.fbS14_AssemblyPost.fbPIM)
        shows AircomLibrary.vStationPIM(fbPIM := MAIN.fbS15_AssemblyPost.fbPIM)
        shows AircomLibrary.vStationPIM(fbPIM := MAIN.fbS16_SonictechUSW.fbPIM)
        shows AircomLibrary.vStationPIM(fbPIM := MAIN.fbS17_SonictechUSW.fbPIM)
        shows AircomLibrary.vStationPIM(fbPIM := MAIN.fbS19_1_EOL3.fbPIM)
        shows AircomLibrary.vStationPIM(fbPIM := MAIN.fbS19_2_EOL3.fbPIM)
        shows AircomLibrary.vStationPIM(fbPIM := MAIN.fbS20_AssemblyPost.fbPIM)
        shows AircomLibrary.vStationPIM(fbPIM := MAIN.fbS21_DetectionTunel.fbPIM)
        shows AircomLibrary.vStationPIM(fbPIM := MAIN.fbS22_SetPackingStation.fbPIM)
        shows AircomLibrary.vStationPIM()
        p2766960713: GVL.fbSqlCore
        p2683556743: GVL.stLJ20_DTL_WorkParams
        p3043078949: MAIN.fbLL19_1_EOL3
        p1709583229: GVL.stLL19_EOL_Settings_I
        p2719655782: MAIN.fbLL19_2_EOL3
        p3094409976: GVL.stLL19_EOL_Settings_II
        p74549115: 'Left chamber'
        p3369830373: 'Right chamber'
        p3445515547: MAIN.fbLS06
        p3589162504: GVL_IO.stLS01_HoseCutter
        p458721708: MAIN.fbLS01_HoseCutter
        p3390713232: MAIN.fbLS04_1_Station
        p1393785898: MAIN.fbLS04_2_Station
        p3419948967: MAIN.fbLS05_1_Station
        p1389434397: MAIN.fbLS05_2_Station
        p422258626: MAIN.fbLS04_1_Crimper
        p417943029: MAIN.fbLS05_1_Crimper
        p2149742200: MAIN.fbLS04_2_Crimper
        p2178948175: MAIN.fbLS05_2_Crimper
        p180551898: MAIN.fbS03
        p2110009420: MAIN.fbLS02_InsertAssy
        p2404496545: MAIN.fbLS02_Station
        p4166419511: MAIN.fbLS03_Station
        p1449093633: MAIN.fbLS06_V2
        p898092448: GVL.Hose_Tester_Params_V2
        p589997586: GVL.Hose_Tester_Params_V2.iPickedHose
        p1762866656: MAIN.fbS03
        p504628598: MAIN.fbLS02_InsertAssy
        p1957019379: MAIN.fbLS06_V2
        p1712759876: GVL.Hose_Tester_Params_V2
        p3689475492: GVL.Hose_Tester_Params_V2.iPickedHose
        p1628323955: MAIN.fbS21_DetectionTunel.fbPIM
        p2913222893: MAIN.fbS22_SetPackingStation.fbPIM
    Rectangle (5,5 140x40), "BH0LPL"
        OnMouseDown: FrameSelectionChange Selection=SelectedFrame=cd818c81-a6c5-4ab8-9515-1ee8055884ac, GlobSel=AssignType=Directly, SelType=Locally
    Rectangle (5,60 140x30), "BH0LPL01_M1"
        OnMouseDown: FrameSelectionChange Selection=SelectedFrame=cd818c81-a6c5-4ab8-9515-1ee8055884ac, Selection=1, GlobSel=AssignType=Directly, SelType=Locally
    Rectangle (5,95 140x30), "BH0LPL01_M2"
        OnMouseDown: FrameSelectionChange Selection=SelectedFrame=cd818c81-a6c5-4ab8-9515-1ee8055884ac, Selection=2, GlobSel=AssignType=Directly, SelType=Locally
    Rectangle (5,130 140x30), "BH0LPL01_M3"
        OnMouseDown: FrameSelectionChange Selection=SelectedFrame=cd818c81-a6c5-4ab8-9515-1ee8055884ac, Selection=3, GlobSel=AssignType=Directly, SelType=Locally
END_VISUALIZATION

// ---- VISUs/New Visus/HomeVisuBH0MPL.TcVIS
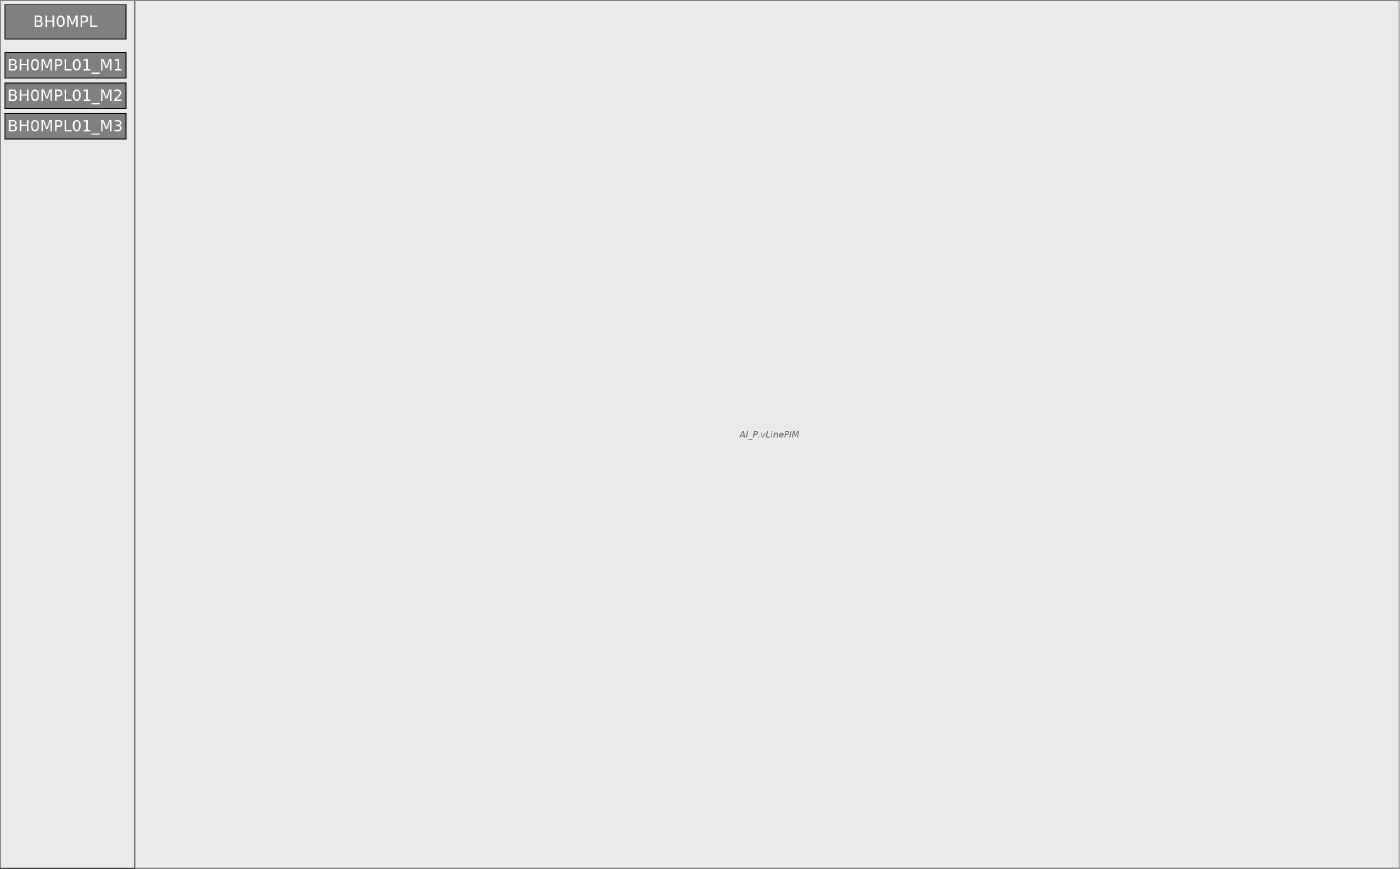
VISUALIZATION HomeVisuBH0MPL  // 1610x1000
    Rectangle (0,0 155x1000)
    Frame (155,0 1460x1000)
        shows AI_P.vLinePIM(fbPIM := MAIN.stLine_BH0MPL.fbLine)
        shows AI_P.vStationPIM(fbPIM := MAIN.fbHotPlate_G7_M1.fbPIM)
        shows AI_P.vStationPIM(fbPIM := MAIN.fbHotPlate_G7_M2.fbPIM)
        shows AI_P.vStationPIM(fbPIM := MAIN.fbHotPlate_G7_M3.fbPIM)
        shows AircomLibrary.vStationPIM(fbPIM := MAIN.fbS14_AssemblyPost.fbPIM)
        shows AircomLibrary.vStationPIM(fbPIM := MAIN.fbS15_AssemblyPost.fbPIM)
        shows AircomLibrary.vStationPIM(fbPIM := MAIN.fbS16_SonictechUSW.fbPIM)
        shows AircomLibrary.vStationPIM(fbPIM := MAIN.fbS17_SonictechUSW.fbPIM)
        shows AircomLibrary.vStationPIM(fbPIM := MAIN.fbS19_1_EOL3.fbPIM)
        shows AircomLibrary.vStationPIM(fbPIM := MAIN.fbS19_2_EOL3.fbPIM)
        shows AircomLibrary.vStationPIM(fbPIM := MAIN.fbS20_AssemblyPost.fbPIM)
        shows AircomLibrary.vStationPIM(fbPIM := MAIN.fbS21_DetectionTunel.fbPIM)
        shows AircomLibrary.vStationPIM(fbPIM := MAIN.fbS22_SetPackingStation.fbPIM)
        shows AircomLibrary.vStationPIM()
        p2766960713: GVL.fbSqlCore
        p2683556743: GVL.stLJ20_DTL_WorkParams
        p3043078949: MAIN.fbLL19_1_EOL3
        p1709583229: GVL.stLL19_EOL_Settings_I
        p2719655782: MAIN.fbLL19_2_EOL3
        p3094409976: GVL.stLL19_EOL_Settings_II
        p74549115: 'Left chamber'
        p3369830373: 'Right chamber'
        p3445515547: MAIN.fbLS06
        p3589162504: GVL_IO.stLS01_HoseCutter
        p458721708: MAIN.fbLS01_HoseCutter
        p3390713232: MAIN.fbLS04_1_Station
        p1393785898: MAIN.fbLS04_2_Station
        p3419948967: MAIN.fbLS05_1_Station
        p1389434397: MAIN.fbLS05_2_Station
        p422258626: MAIN.fbLS04_1_Crimper
        p417943029: MAIN.fbLS05_1_Crimper
        p2149742200: MAIN.fbLS04_2_Crimper
        p2178948175: MAIN.fbLS05_2_Crimper
        p180551898: MAIN.fbS03
        p2110009420: MAIN.fbLS02_InsertAssy
        p2404496545: MAIN.fbLS02_Station
        p4166419511: MAIN.fbLS03_Station
        p1449093633: MAIN.fbLS06_V2
        p898092448: GVL.Hose_Tester_Params_V2
        p589997586: GVL.Hose_Tester_Params_V2.iPickedHose
        p1762866656: MAIN.fbS03
        p504628598: MAIN.fbLS02_InsertAssy
        p1957019379: MAIN.fbLS06_V2
        p1712759876: GVL.Hose_Tester_Params_V2
        p3689475492: GVL.Hose_Tester_Params_V2.iPickedHose
        p1628323955: MAIN.fbS21_DetectionTunel.fbPIM
        p2913222893: MAIN.fbS22_SetPackingStation.fbPIM
    Rectangle (5,5 140x40), "BH0MPL"
        OnMouseDown: FrameSelectionChange Selection=SelectedFrame=cd818c81-a6c5-4ab8-9515-1ee8055884ac, GlobSel=AssignType=Directly, SelType=Locally
    Rectangle (5,60 140x30), "BH0MPL01_M1"
        OnMouseDown: FrameSelectionChange Selection=SelectedFrame=cd818c81-a6c5-4ab8-9515-1ee8055884ac, Selection=1, GlobSel=AssignType=Directly, SelType=Locally
    Rectangle (5,95 140x30), "BH0MPL01_M2"
        OnMouseDown: FrameSelectionChange Selection=SelectedFrame=cd818c81-a6c5-4ab8-9515-1ee8055884ac, Selection=2, GlobSel=AssignType=Directly, SelType=Locally
    Rectangle (5,130 140x30), "BH0MPL01_M3"
        OnMouseDown: FrameSelectionChange Selection=SelectedFrame=cd818c81-a6c5-4ab8-9515-1ee8055884ac, Selection=3, GlobSel=AssignType=Directly, SelType=Locally
END_VISUALIZATION

// ---- VISUs/New Visus/HomeVisuBO02PL.TcVIS
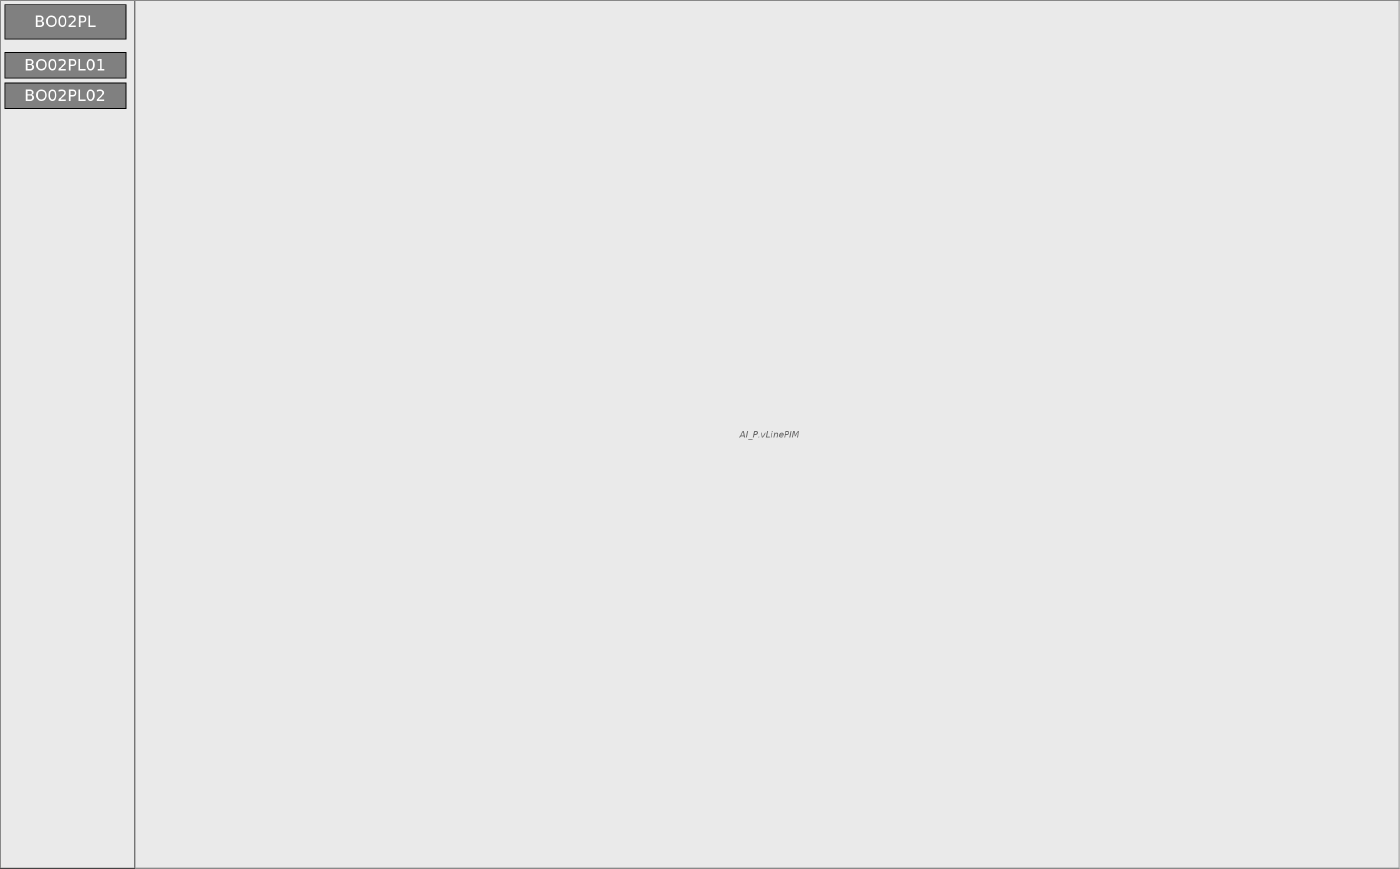
VISUALIZATION HomeVisuBO02PL  // 1610x1000
    Rectangle (0,0 155x1000)
    Frame (155,0 1460x1000)
        shows AI_P.vLinePIM(fbPIM := MAIN.stLine_BO02PL.fbLine)
        shows AI_P.vStationPIM(fbPIM := MAIN.fbS03_BearingPress.fbPIM)
        shows AI_P.vStationPIM(fbPIM := MAIN.fbS04_BearingPress.fbPIM)
        shows AircomLibrary.vStationPIM(fbPIM := MAIN.fbS13_FrontFan.fbPIM)
        shows AircomLibrary.vStationPIM(fbPIM := MAIN.fbS14_AssemblyPost.fbPIM)
        shows AircomLibrary.vStationPIM(fbPIM := MAIN.fbS15_AssemblyPost.fbPIM)
        shows AircomLibrary.vStationPIM(fbPIM := MAIN.fbS16_SonictechUSW.fbPIM)
        shows AircomLibrary.vStationPIM(fbPIM := MAIN.fbS17_SonictechUSW.fbPIM)
        shows AircomLibrary.vStationPIM(fbPIM := MAIN.fbS19_1_EOL3.fbPIM)
        shows AircomLibrary.vStationPIM(fbPIM := MAIN.fbS19_2_EOL3.fbPIM)
        shows AircomLibrary.vStationPIM(fbPIM := MAIN.fbS20_AssemblyPost.fbPIM)
        shows AircomLibrary.vStationPIM(fbPIM := MAIN.fbS21_DetectionTunel.fbPIM)
        shows AircomLibrary.vStationPIM(fbPIM := MAIN.fbS22_SetPackingStation.fbPIM)
        shows AircomLibrary.vStationPIM()
        p2766960713: GVL.fbSqlCore
        p2683556743: GVL.stLJ20_DTL_WorkParams
        p3043078949: MAIN.fbLL19_1_EOL3
        p1709583229: GVL.stLL19_EOL_Settings_I
        p2719655782: MAIN.fbLL19_2_EOL3
        p3094409976: GVL.stLL19_EOL_Settings_II
        p74549115: 'Left chamber'
        p3369830373: 'Right chamber'
        p3445515547: MAIN.fbLS06
        p3589162504: GVL_IO.stLS01_HoseCutter
        p458721708: MAIN.fbLS01_HoseCutter
        p3390713232: MAIN.fbLS04_1_Station
        p1393785898: MAIN.fbLS04_2_Station
        p3419948967: MAIN.fbLS05_1_Station
        p1389434397: MAIN.fbLS05_2_Station
        p422258626: MAIN.fbLS04_1_Crimper
        p417943029: MAIN.fbLS05_1_Crimper
        p2149742200: MAIN.fbLS04_2_Crimper
        p2178948175: MAIN.fbLS05_2_Crimper
        p180551898: MAIN.fbS03
        p2110009420: MAIN.fbLS02_InsertAssy
        p2404496545: MAIN.fbLS02_Station
        p4166419511: MAIN.fbLS03_Station
        p1449093633: MAIN.fbLS06_V2
        p898092448: GVL.Hose_Tester_Params_V2
        p589997586: GVL.Hose_Tester_Params_V2.iPickedHose
        p1762866656: MAIN.fbS03
        p504628598: MAIN.fbLS02_InsertAssy
        p1957019379: MAIN.fbLS06_V2
        p1712759876: GVL.Hose_Tester_Params_V2
        p3689475492: GVL.Hose_Tester_Params_V2.iPickedHose
        p1628323955: MAIN.fbS21_DetectionTunel.fbPIM
        p2913222893: MAIN.fbS22_SetPackingStation.fbPIM
    Rectangle (5,5 140x40), "BO02PL"
        OnMouseDown: FrameSelectionChange Selection=SelectedFrame=cd818c81-a6c5-4ab8-9515-1ee8055884ac, GlobSel=AssignType=Directly, SelType=Locally
    Rectangle (5,60 140x30), "BO02PL01"
        OnMouseDown: FrameSelectionChange Selection=SelectedFrame=cd818c81-a6c5-4ab8-9515-1ee8055884ac, Selection=1, GlobSel=AssignType=Directly, SelType=Locally
    Rectangle (5,95 140x30), "BO02PL02"
        OnMouseDown: FrameSelectionChange Selection=SelectedFrame=cd818c81-a6c5-4ab8-9515-1ee8055884ac, Selection=2, GlobSel=AssignType=Directly, SelType=Locally
END_VISUALIZATION

// ---- VISUs/New Visus/HomeVisuBS02PL.TcVIS
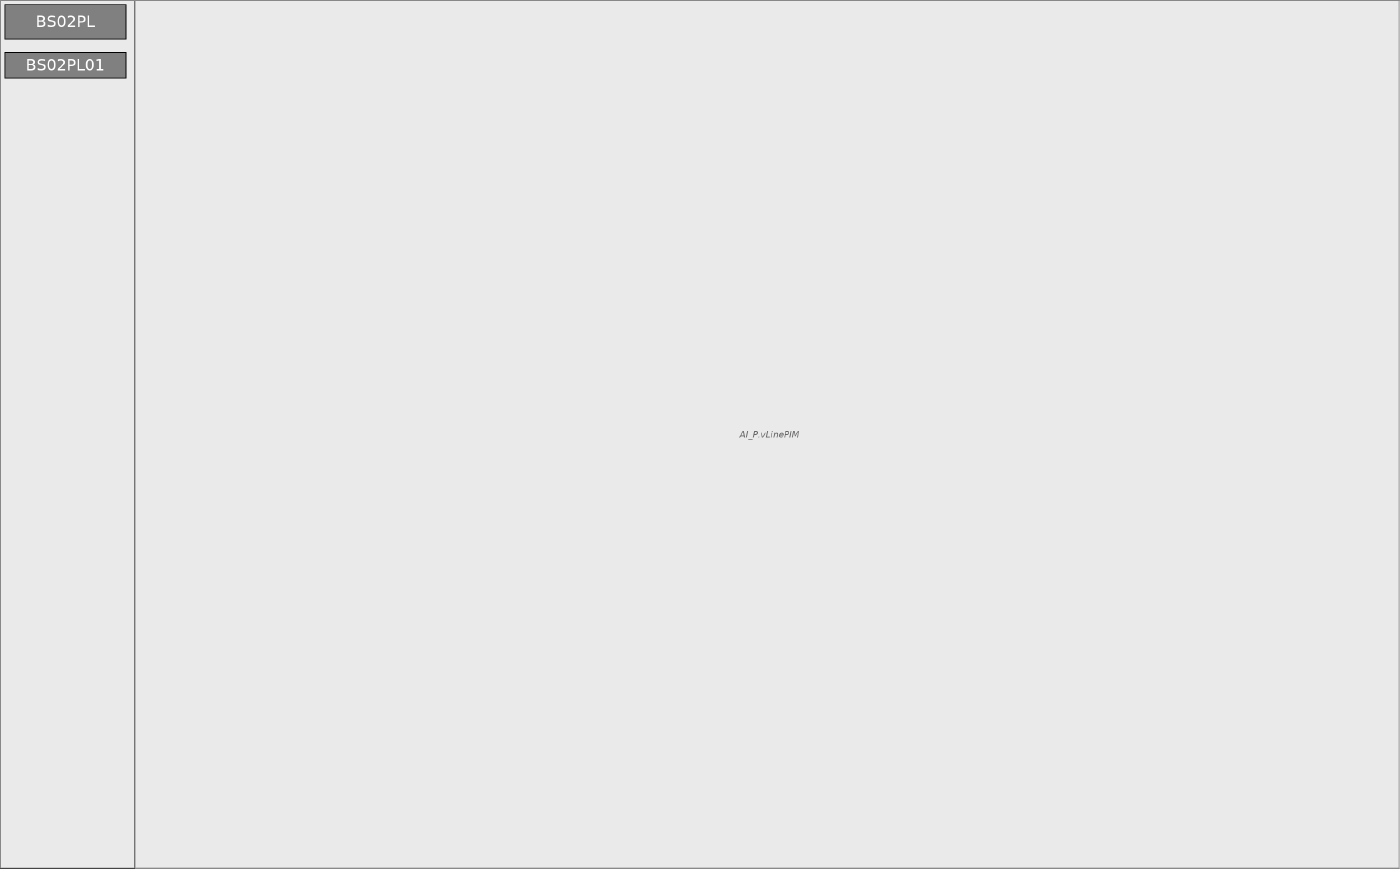
VISUALIZATION HomeVisuBS02PL  // 1610x1000
    Rectangle (0,0 155x1000)
    Frame (155,0 1460x1000)
        shows AI_P.vLinePIM(fbPIM := MAIN.stLine_BS02PL.fbLine)
        shows AI_P.vStationPIM(fbPIM := MAIN.fbS01_BearingPress.fbPIM)
        shows AircomLibrary.vStationPIM(fbPIM := MAIN.fbS13_FrontFan.fbPIM)
        shows AircomLibrary.vStationPIM(fbPIM := MAIN.fbS14_AssemblyPost.fbPIM)
        shows AircomLibrary.vStationPIM(fbPIM := MAIN.fbS12_Hios.fbPIM)
        shows AircomLibrary.vStationPIM(fbPIM := MAIN.fbS15_AssemblyPost.fbPIM)
        shows AircomLibrary.vStationPIM(fbPIM := MAIN.fbS16_SonictechUSW.fbPIM)
        shows AircomLibrary.vStationPIM(fbPIM := MAIN.fbS17_SonictechUSW.fbPIM)
        shows AircomLibrary.vStationPIM(fbPIM := MAIN.fbS19_1_EOL3.fbPIM)
        shows AircomLibrary.vStationPIM(fbPIM := MAIN.fbS19_2_EOL3.fbPIM)
        shows AircomLibrary.vStationPIM(fbPIM := MAIN.fbS20_AssemblyPost.fbPIM)
        shows AircomLibrary.vStationPIM(fbPIM := MAIN.fbS21_DetectionTunel.fbPIM)
        shows AircomLibrary.vStationPIM(fbPIM := MAIN.fbS22_SetPackingStation.fbPIM)
        shows AircomLibrary.vStationPIM()
        p2766960713: GVL.fbSqlCore
        p2683556743: GVL.stLJ20_DTL_WorkParams
        p3043078949: MAIN.fbLL19_1_EOL3
        p1709583229: GVL.stLL19_EOL_Settings_I
        p2719655782: MAIN.fbLL19_2_EOL3
        p3094409976: GVL.stLL19_EOL_Settings_II
        p74549115: 'Left chamber'
        p3369830373: 'Right chamber'
        p3445515547: MAIN.fbLS06
        p3589162504: GVL_IO.stLS01_HoseCutter
        p458721708: MAIN.fbLS01_HoseCutter
        p3390713232: MAIN.fbLS04_1_Station
        p1393785898: MAIN.fbLS04_2_Station
        p3419948967: MAIN.fbLS05_1_Station
        p1389434397: MAIN.fbLS05_2_Station
        p422258626: MAIN.fbLS04_1_Crimper
        p417943029: MAIN.fbLS05_1_Crimper
        p2149742200: MAIN.fbLS04_2_Crimper
        p2178948175: MAIN.fbLS05_2_Crimper
        p180551898: MAIN.fbS03
        p2110009420: MAIN.fbLS02_InsertAssy
        p2404496545: MAIN.fbLS02_Station
        p4166419511: MAIN.fbLS03_Station
        p1449093633: MAIN.fbLS06_V2
        p898092448: GVL.Hose_Tester_Params_V2
        p589997586: GVL.Hose_Tester_Params_V2.iPickedHose
        p1762866656: MAIN.fbS03
        p504628598: MAIN.fbLS02_InsertAssy
        p1957019379: MAIN.fbLS06_V2
        p1712759876: GVL.Hose_Tester_Params_V2
        p3689475492: GVL.Hose_Tester_Params_V2.iPickedHose
        p1628323955: MAIN.fbS21_DetectionTunel.fbPIM
        p2913222893: MAIN.fbS22_SetPackingStation.fbPIM
    Rectangle (5,5 140x40), "BS02PL"
        OnMouseDown: FrameSelectionChange Selection=SelectedFrame=cd818c81-a6c5-4ab8-9515-1ee8055884ac, GlobSel=AssignType=Directly, SelType=Locally
    Rectangle (5,60 140x30), "BS02PL01"
        OnMouseDown: FrameSelectionChange Selection=SelectedFrame=cd818c81-a6c5-4ab8-9515-1ee8055884ac, Selection=1, GlobSel=AssignType=Directly, SelType=Locally
END_VISUALIZATION

// ---- VISUs/New Visus/HomeVisu_1.TcVIS
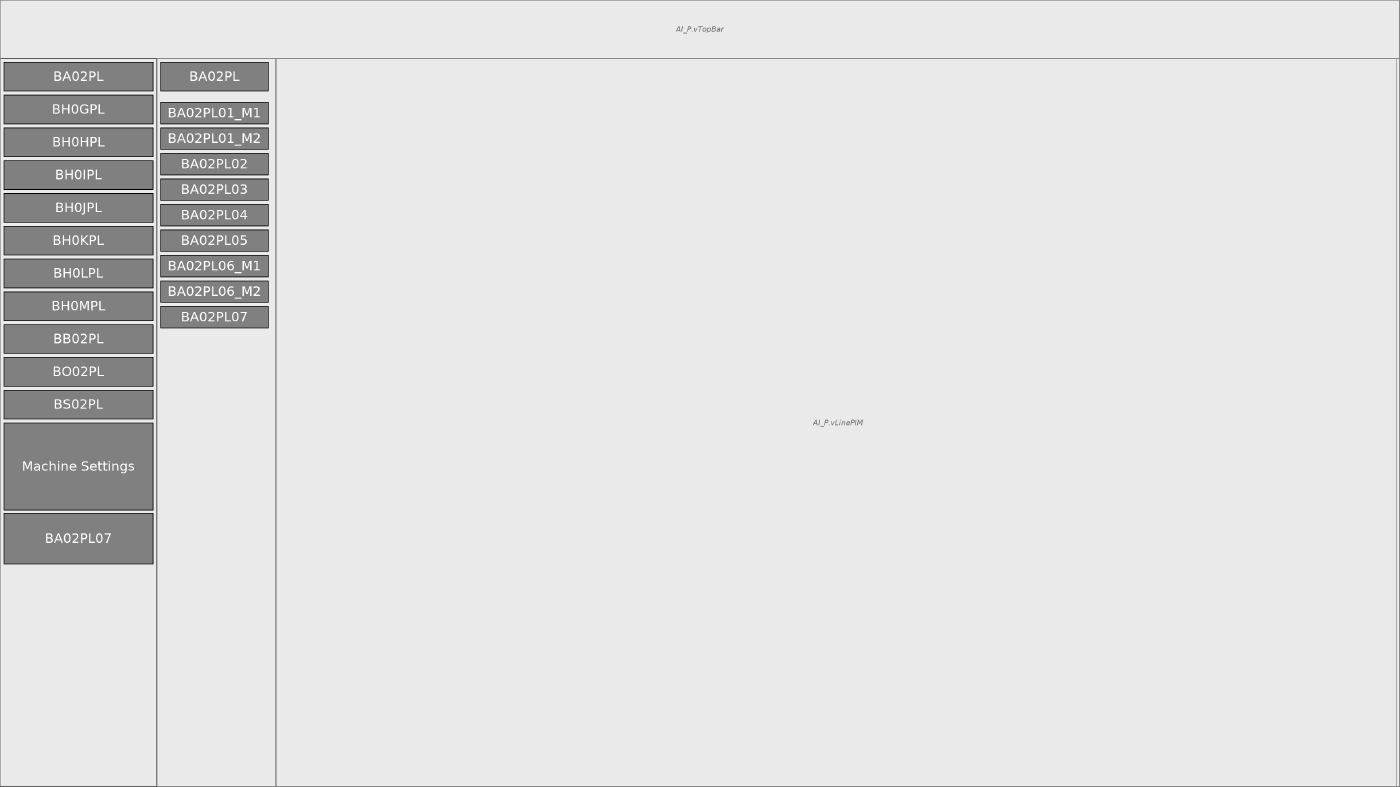
VISUALIZATION HomeVisu_1  // 1920x1080
    Rectangle (0,80 215x1000)
    Frame (215,80 1700x1000)
        shows HomeVisuBA02PL()
        shows HomeVisuBH0GPL()
        shows HomeVisuBH0HPL()
        shows HomeVisuBH0IPL()
        shows HomeVisuBH0JPL()
        shows HomeVisuBH0KPL()
        shows HomeVisuBH0LPL()
        shows HomeVisuBH0MPL()
        shows HomeVisuBB02PL()
        shows HomeVisuBO02PL()
        shows HomeVisuBS02PL()
        shows vHotPlateSettings_V3_B02PL(fbHP1_M1 := MAIN.fbHotPlate_G1_M1, fbHP1_M2 := MAIN.fbHotPlate_G1_M2, fbHP1_M3 := MAIN.fbHotPlate_G1_M3, fbHP2_M1 := MAIN.fbHotPlate_G2_M1, fbHP2_M2 := MAIN.fbHotPlate_G2_M2, fbHP2_M3 := MAIN.fbHotPlate_G2_M3, fbHP3_M1 := MAIN.fbHotPlate_G3_M1, fbHP3_M2 := MAIN.fbHotPlate_G3_M2, fbHP3_M3 := MAIN.fbHotPlate_G3_M3, fbHP4_M1 := MAIN.fbHotPlate_G4_M1, fbHP4_M2 := MAIN.fbHotPlate_G4_M2, fbHP4_M3 := MAIN.fbHotPlate_G4_M3, fbHP5_M1 := MAIN.fbHotPlate_G5_M1, fbHP5_M2 := MAIN.fbHotPlate_G5_M2, fbHP5_M3 := MAIN.fbHotPlate_G5_M3, fbHP6_M1 := MAIN.fbHotPlate_G6_M1, fbHP6_M2 := MAIN.fbHotPlate_G6_M2, fbHP6_M3 := MAIN.fbHotPlate_G6_M3, fbHP7_M1 := MAIN.fbHotPlate_G7_M1, fbHP7_M2 := MAIN.fbHotPlate_G7_M2, fbHP7_M3 := MAIN.fbHotPlate_G7_M3, fbS01_Press := MAIN.fbS01_BearingPress, fbS01_FixtureBase := MAIN.fbS01_KeyencePNVisSens, fbS02_Press := MAIN.fbS02_BearingPress, fbS03_Press := MAIN.fbS03_BearingPress, fbS03_FixtureBase := MAIN.fbS03_CapFixture, fbS04_Press := MAIN.fbS04_BearingPress, stHMIData_Filler_A := MAIN.fb_Filler_A_Machine.stHMI, stParams_Filler_A := MAIN.fb_Filler_A_Machine.stSlaveParms, stHMIData_Cork := MAIN.fb_Cork_Machine.stHMI, stParams_Cork := MAIN.fb_Cork_Machine.stSlaveParms, stHMIData_Filler_B := MAIN.fb_Filler_B_Machine.stHMI, stParams_Filler_B := MAIN.fb_Filler_B_Machine.stSlaveParms, stHMIData_Sticker := MAIN.fb_Sticker_Machine.stHMI, stParams_Sticker := MAIN.fb_Sticker_Machine.stSlaveParms, stHMIData_Laser := MAIN.fb_Laser_Machine.stHMI, stParams_Laser := MAIN.fb_Laser_Machine.stSlaveParms, stHMI_Laser := MAIN.fb_Laser_Machine.fbLaserControl.stHMI_Laser, fbSonic_S02 := MAIN.fb_1_SonicTech_SonictechUSW, fbSonic_S04 := MAIN.fb_2_SonicTech_SonictechUSW, fbVacuumChamber := MAIN.fb_UnderPressure_Tester_Machine, fbTransporter := MAIN.fbTransporterUnderpressure)
        shows AI_M.vWeighingTunnel(fbWeighingTunel := MAIN.fbWeighingTunel)
        shows vWeighingTunelVisionFrame()
        shows vStations19_21_22()
        p3043078949: MAIN.fbLL19_1_EOL3
        p1709583229: GVL.stLL19_EOL_Settings_I
        p2719655782: MAIN.fbLL19_2_EOL3
        p3094409976: GVL.stLL19_EOL_Settings_II
        p74549115: 'Left chamber'
        p3369830373: 'Right chamber'
        p4001053958: MAIN.fbS21_DetectionTunel
        p3623223747: MAIN.fbS21_DetectionTunel
        p3171485557: GVL.stS21_DTL_WorkParams
        p817651737: MAIN.stStation_LCA01PL_SCA01PL21
        p3449029454: GVL.stS21_DTL_Settings
        p3777340465: MAIN.fbS19_RecipeManager
        p3453682166: MAIN.stS19_EOL3_TMP_TestParams
        p3169997168: GVL_IO.stS21_DTL_InOuts.iLaserCurrentValue
        p2878062980: MAIN.fbS11_ResWelder.fbPIM
        p847417406: MAIN.fbS12_HiosScrewDriver.fbPIM
        p1166385320: MAIN.fbS13_FrontFanPress.fbPIM
        p3688969483: MAIN.fbS14_AssemblyPostCtrl.fbPIM
        p2900755869: MAIN.fbS15_AssemblyPostCtrl.fbPIM
        p3528948000: MAIN.fbS18_LabelSticking.fbPIM
        p514386723: MAIN.fbS22_SetPackingStation
        p2740858475: MAIN.fbS18_LabelSticking.stInOuts.iPressure
        p901175331: MAIN.fbS18_LabelSticking.stTestParams
        p1258792094: MAIN.fbS15_AssemblyPostCtrl.stWorkParams
        p1006670856: MAIN.fbS14_AssemblyPostCtrl.stWorkParams
        p2724463019: MAIN.fbS13_FrontFanPress.stParams
        p3580047677: MAIN.fbS12_HiosScrewDriver.stTestParam
        p1282039943: MAIN.fbS11_ResWelder.stWorkParams
        p285620971: GVL.stS19_EOL_TestParams
        p2487237938: MAIN.fbS19_1_EOL3
        p1850671185: MAIN.fbS19_2_EOL3
        p4100169850: GVL.stS19_EOL_Settings_I
        p241999129: GVL.stS19_EOL_Settings_II
        p1128139719: MAIN.fbS11_ResWelder.fbPIM
        p3661060733: MAIN.fbS12_HiosScrewDriver.fbPIM
        p2905631467: MAIN.fbS13_FrontFanPress.fbPIM
        p861208392: MAIN.fbS14_AssemblyPostCtrl.fbPIM
        p1146343390: MAIN.fbS15_AssemblyPostCtrl.fbPIM
        p987935587: MAIN.fbS18_LabelSticking.fbPIM
        p3446969237: GVL.stS18_ManometerCalibration_TestData
        p715956300: GVL.stS18_PressureScalingData
        p3016093480: GVL.stS15_AssemblyPostParams
        p3301105598: GVL.stS14_AssemblyPostParams
        p1520847389: GVL.stS13_Parameters
        p765557387: GVL.stS12_Parameters
        p3030919985: MAIN.fbS11_ResWelder.stWorkParams
        p4053094083: MAIN.fbS22_SetPackingStation
        p662549438: MAIN.fbS18_LabelSticking.stInOuts.iPressure
        p2928623001: GVL.stS18_PressureScalingData
        p1931357957: MAIN.fbS01_SonictechUSW.fbPIM
        p2635091497: MAIN.fbS03_SonictechUSW.fbPIM
        p1953753884: MAIN.fbS05_1_SonictechUSW.fbPIM
        p3984243366: MAIN.fbS06_SonictechUSW.fbPIM
        p2591918640: MAIN.fbS07_SonictechUSW.fbPIM
        p180524961: MAIN.fbS08_SonictechUSW.fbPIM
        p2110105399: MAIN.fbS09_SonictechUSW.fbPIM
        p486682322: MAIN.fbS10_SonictechUSW.fbPIM
        p4100033511: MAIN.fbS16_SonictechUSW.fbPIM
        p2204547953: MAIN.fbS17_SonictechUSW.fbPIM
        p3358502448: MAIN.fbS07_FixCarrierPistonAssy.stInOuts.rHeatStampTemperature
        p3363745968: GVL.stS01_FixSettings
        p644927900: GVL.stS03_FixSettings
        p3474158761: GVL.stS05_BallPressSettings
        p2347394456: GVL.stS05_USWelderSettings
        p1444554003: GVL.stS06_FixSettings
        p555554181: GVL.stS07_FixSettings
        p2980186132: GVL.stS08_FixSettings
        p3332716674: GVL.stS09_USWelderSettings
        p2791485799: GVL.stS10_USWelderSettings
        p1325470802: GVL.stS16_FixSettings
        p939926724: GVL.stS17_FixSettings
        p2967930134: GVL.stS21_DTL_Settings
        p2380948999: GVL_IO.stS21_DTL_InOuts.iLaserCurrentValue
        p3200496103: MAIN.fb_UnderPressure_Tester_Machine.stInOuts
        p980272329: MAIN.fb_UnderPressure_Tester_Machine.stParams
        p182610665: MAIN.fb_UnderPressure_Tester_Machine.stStatus
        p3000099066: MAIN.fb_UnderPressure_Tester_Machine.iWorkStep
        p1064606418: MAIN.fbTransporterUnderpressure.stInOuts
        p3808140917: MAIN.fbTransporterUnderpressure.stStatus
        p1825866306: MAIN.fbTransporterUnderpressure.iWorkStep
    Frame (0,0 1920x80)
        shows AI_P.vTopBar(fbLine := MAIN.stLine_BA02PL.fbLine)
    Rectangle (5,85 205x40), "BA02PL"
        OnMouseDown: FrameSelectionChange Selection=SelectedFrame=6c9ea511-e956-4d78-8ee8-89cc4cfbd0e1, GlobSel=AssignType=Directly, SelType=Locally
    Rectangle (5,130 205x40), "BH0GPL"
        OnMouseDown: FrameSelectionChange Selection=SelectedFrame=6c9ea511-e956-4d78-8ee8-89cc4cfbd0e1, Selection=1, GlobSel=AssignType=Directly, SelType=Locally
    Rectangle (5,580 205x120), "Machine Settings"
        OnMouseDown: FrameSelectionChange Selection=SelectedFrame=6c9ea511-e956-4d78-8ee8-89cc4cfbd0e1, Selection=11, GlobSel=AssignType=Directly, SelType=Locally
    Rectangle (5,175 205x40), "BH0HPL"
        OnMouseDown: FrameSelectionChange Selection=SelectedFrame=6c9ea511-e956-4d78-8ee8-89cc4cfbd0e1, Selection=2, GlobSel=AssignType=Directly, SelType=Locally
    Rectangle (5,265 205x40), "BH0JPL"
        OnMouseDown: FrameSelectionChange Selection=SelectedFrame=6c9ea511-e956-4d78-8ee8-89cc4cfbd0e1, Selection=4, GlobSel=AssignType=Directly, SelType=Locally
    Rectangle (5,220 205x40), "BH0IPL"
        OnMouseDown: FrameSelectionChange Selection=SelectedFrame=6c9ea511-e956-4d78-8ee8-89cc4cfbd0e1, Selection=3, GlobSel=AssignType=Directly, SelType=Locally
    Rectangle (5,310 205x40), "BH0KPL"
        OnMouseDown: FrameSelectionChange Selection=SelectedFrame=6c9ea511-e956-4d78-8ee8-89cc4cfbd0e1, Selection=5, GlobSel=AssignType=Directly, SelType=Locally
    Rectangle (5,355 205x40), "BH0LPL"
        OnMouseDown: FrameSelectionChange Selection=SelectedFrame=6c9ea511-e956-4d78-8ee8-89cc4cfbd0e1, Selection=6, GlobSel=AssignType=Directly, SelType=Locally
    Rectangle (5,445 205x40), "BB02PL"
        OnMouseDown: FrameSelectionChange Selection=SelectedFrame=6c9ea511-e956-4d78-8ee8-89cc4cfbd0e1, Selection=8, GlobSel=AssignType=Directly, SelType=Locally
    Rectangle (5,400 205x40), "BH0MPL"
        OnMouseDown: FrameSelectionChange Selection=SelectedFrame=6c9ea511-e956-4d78-8ee8-89cc4cfbd0e1, Selection=7, GlobSel=AssignType=Directly, SelType=Locally
    Rectangle (5,490 205x40), "BO02PL"
        OnMouseDown: FrameSelectionChange Selection=SelectedFrame=6c9ea511-e956-4d78-8ee8-89cc4cfbd0e1, Selection=9, GlobSel=AssignType=Directly, SelType=Locally
    Rectangle (5,535 205x40), "BS02PL"
        OnMouseDown: FrameSelectionChange Selection=SelectedFrame=6c9ea511-e956-4d78-8ee8-89cc4cfbd0e1, Selection=10, GlobSel=AssignType=Directly, SelType=Locally
    Rectangle (5,704 205x70), "BA02PL07"
        OnMouseDown: FrameSelectionChange Selection=SelectedFrame=6c9ea511-e956-4d78-8ee8-89cc4cfbd0e1, Selection=12, GlobSel=AssignType=Directly, SelType=Locally
END_VISUALIZATION

// ---- VISUs/New Visus/vHotPlateSettings_V3_B02PL.TcVIS
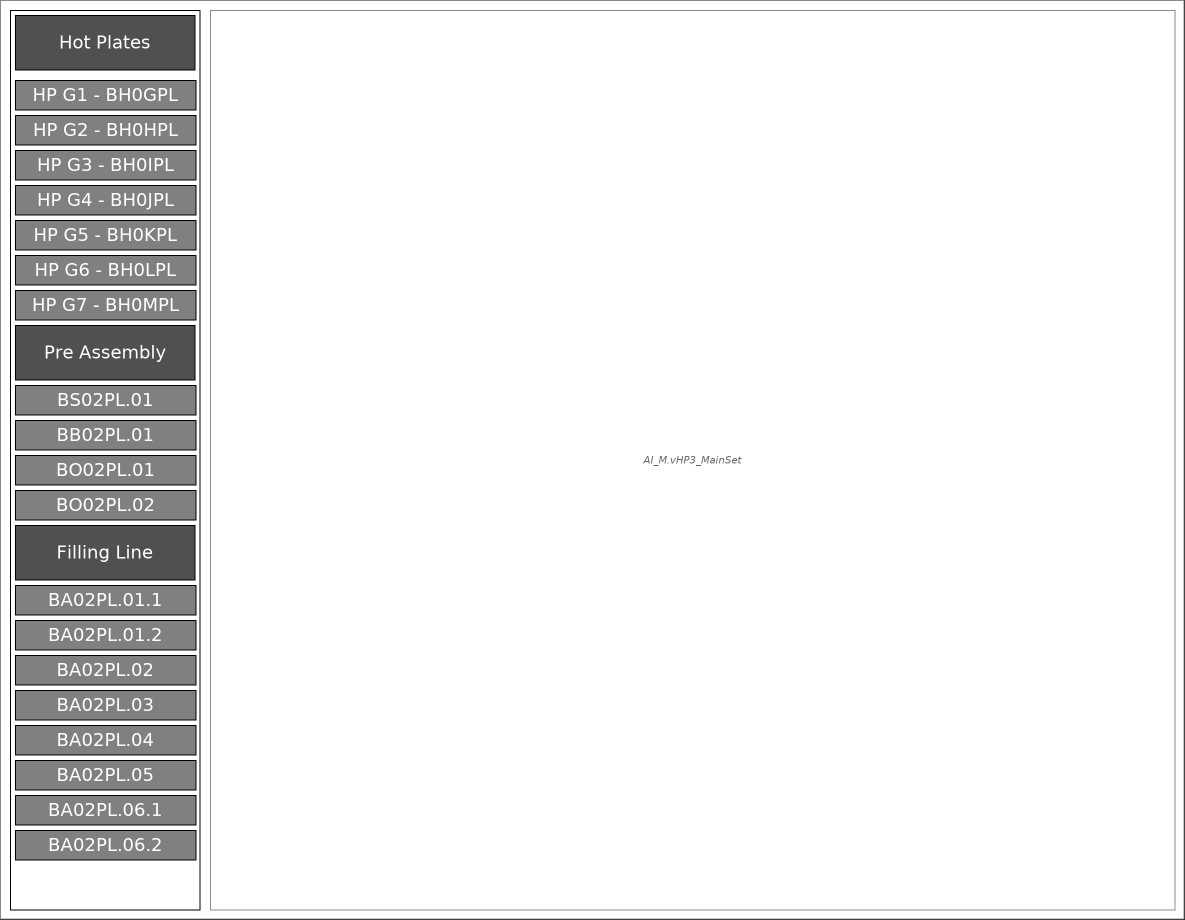
VISUALIZATION vHotPlateSettings_V3_B02PL  // 1185x920
VAR_IN_OUT
	fbHP1_M1	: fbHP_Control_V3_1;
	fbHP1_M2	: fbHP_Control_V3_1;
	fbHP1_M3	: fbHP_Control_V3_1;
	
	fbHP2_M1	: fbHP_Control_V3_1;
	fbHP2_M2	: fbHP_Control_V3_1;
	fbHP2_M3	: fbHP_Control_V3_1;
	
	fbHP3_M1	: fbHP_Control_V3_1;
	fbHP3_M2	: fbHP_Control_V3_1;
	fbHP3_M3	: fbHP_Control_V3_1;
	
	fbHP4_M1	: fbHP_Control_V3_1;
	fbHP4_M2	: fbHP_Control_V3_1;
	fbHP4_M3	: fbHP_Control_V3_1;
	
	fbHP5_M1	: fbHP_Control_V3_1;
	fbHP5_M2	: fbHP_Control_V3_1;
	fbHP5_M3	: fbHP_Control_V3_1;
	
	fbHP6_M1	: fbHP_Control_V3_1;
	fbHP6_M2	: fbHP_Control_V3_1;
	fbHP6_M3	: fbHP_Control_V3_1;
	
	fbHP7_M1	: fbHP_Control_V3_1;
	fbHP7_M2	: fbHP_Control_V3_1;
	fbHP7_M3	: fbHP_Control_V3_1;
	
	fbS01_Press						: fbSonicPress_V4_1;
	fbS01_FixtureBase				: fbSealingCorkAssKeyencePN_V4_1;
	
	fbS02_Press						: fbSonicPress_V4_1;
	
	fbS03_Press						: fbSonicPress_V4_1;
	fbS03_FixtureBase				: fbCapDetectionFixture_V4_1;
	
	fbS04_Press						: fbSonicPress_V4_1;
	
	stHMIData_Filler_A				:	stChiniseMachineHmiData_V3_1;
	stParams_Filler_A				:	stModTcpSlaveParams_V3_1;
	
	stHMIData_Cork					:	stChiniseMachineHmiData_V3_1;
	stParams_Cork					:	stModTcpSlaveParams_V3_1;
	
	stHMIData_Filler_B				:	stChiniseMachineHmiData_V3_1;
	stParams_Filler_B				:	stModTcpSlaveParams_V3_1;
	
	stHMIData_Sticker				:	stChiniseMachineHmiData_V3_1;
	stParams_Sticker				:	stModTcpSlaveParams_V3_1;
	
	stHMIData_Laser					:	stChiniseMachineHmiData_V3_2;
	stParams_Laser					:	stModTcpSlaveParams_V3_2;
	stHMI_Laser						: 	stHMI_Laser;
	
	fbSonic_S02						: fbSonictechUSWM_V4_1;
	
	fbSonic_S04						: fbSonictechUSWM_V4_1;
	
	fbVacuumChamber					: fbVacuumChamber_V3_2;
	fbTransporter					: fbTransporter_V3_2;
END_VAR
    Rectangle (0,0 1185x920)
    Frame (210,10 965x900)
        shows AI_M.vHP3_MainSet(fbHP_M1 := fbHP1_M1, fbHP_M2 := fbHP1_M2, fbHP_M3 := fbHP1_M3, NestNumber := 1, sSocketName := 'BH0GPL')
        shows AI_M.vHP3_MainSet(fbHP_M1 := fbHP2_M1, fbHP_M2 := fbHP2_M2, fbHP_M3 := fbHP2_M3, NestNumber := 2, sSocketName := 'BH0HPL')
        shows AI_M.vHP3_MainSet(fbHP_M1 := fbHP3_M1, fbHP_M2 := fbHP3_M2, fbHP_M3 := fbHP3_M3, NestNumber := 3, sSocketName := 'BH0IPL')
        shows AI_M.vHP3_MainSet(fbHP_M1 := fbHP4_M1, fbHP_M2 := fbHP4_M2, fbHP_M3 := fbHP4_M3, NestNumber := 4, sSocketName := 'BH0JPL')
        shows AI_M.vHP3_MainSet(fbHP_M1 := fbHP5_M1, fbHP_M2 := fbHP5_M2, fbHP_M3 := fbHP5_M3, NestNumber := 5, sSocketName := 'BH0KPL')
        shows AI_M.vHP3_MainSet(fbHP_M1 := fbHP6_M1, fbHP_M2 := fbHP6_M2, fbHP_M3 := fbHP6_M3, NestNumber := 6, sSocketName := 'BH0LPL')
        shows AI_M.vHP3_MainSet(fbHP_M1 := fbHP7_M1, fbHP_M2 := fbHP7_M2, fbHP_M3 := fbHP7_M3, NestNumber := 7, sSocketName := 'BH0MPL')
        shows AI_M.vSealingCorkAssPress_V4_1(fbData := fbS01_Press, fbFixtureBase := fbS01_FixtureBase)
        shows AI_M.vBaseSonicTechPress_V4_1(fbData := fbS02_Press)
        shows AI_M.vCapDetectionFixPress_V4_1(fbData := fbS03_Press, fbFixtureBase := fbS03_FixtureBase)
        shows AI_M.vBaseSonicTechPress_V4_1(fbData := fbS04_Press)
        shows AI_M.vChiniseMachineStatus_v3_1(stData := stHMIData_Filler_A, stParams := stParams_Filler_A)
        shows AI_M.vChiniseMachineStatus_v3_1(stData := stHMIData_Cork, stParams := stParams_Cork)
        shows AI_M.vBaseSonicTech_V4_1(fbData := fbSonic_S02)
        shows AI_M.vChiniseMachineStatus_v3_1(stData := stHMIData_Filler_B, stParams := stParams_Filler_B)
        shows AI_M.vBaseSonicTech_V4_1(fbData := fbSonic_S04)
        shows AI_M.vVacuumChamberMain_V3_2(fb := fbVacuumChamber, fbTrans := fbTransporter)
        shows AI_M.vChiniseMachineStatus_v3_1(stData := stHMIData_Sticker, stParams := stParams_Sticker)
        shows AI_M.vChiniseMachineStatus_Laser_V3_2(stData := stHMIData_Laser, stParams := stParams_Laser, stHMI_Laser := stHMI_Laser)
        shows vSetPacking_V3_Status_V3_2(fbData := fbS22)
        shows vDetectionTunelFrame_V3_1(stInOuts := stInOuts_Tunel, stParams := stParams_Tunel, iWorkStep := iWorkStep_Tunel, fb := fb_Tunel)
        p544952995: rS07HeaterTemperature
        p3767341414: fbS20
        p4018227088: fbS18.fbPIM
        p1625067722: fbS18.stHwSettings
        p4124004121: fbS18.stInOuts.iPressure
        p961079038: fbS16.stInOuts
        p1151590893: fbSonic_S16
        p2539462775: fbS14
        p3846459017: fbS11.fbPIM
        p39883683: fbS10
        p445293019: fbSonic_S10
        p2875566315: fbS10.stInOuts
        p426879848: fbSonic_S09.fbPIM.stStation.sStationName
        p268622539: fbS06.stSettings
        p836702480: fbS06.stInOuts
        p773328817: fbSonic_S06.stDigitalInOut
        p11944277: fbSonic_S06
        p847402520: fbS07.stInOuts.rHeatStampTemperature
    Rectangle (10,10 190x900)
    Rectangle (15,80 181x30), "HP G1 - BH0GPL"
        OnMouseDown: FrameSelectionChange Selection=SelectedFrame=2676ba61-b932-4ea5-9074-f1d3beec8c67, GlobSel=AssignType=Directly, SelType=Locally
    Rectangle (15,15 180x55), "Hot Plates"
    Rectangle (15,115 181x30), "HP G2 - BH0HPL"
        OnMouseDown: FrameSelectionChange Selection=SelectedFrame=2676ba61-b932-4ea5-9074-f1d3beec8c67, Selection=1, GlobSel=AssignType=Directly, SelType=Locally
    Rectangle (15,255 181x30), "HP G6 - BH0LPL"
        OnMouseDown: FrameSelectionChange Selection=SelectedFrame=2676ba61-b932-4ea5-9074-f1d3beec8c67, Selection=5, GlobSel=AssignType=Directly, SelType=Locally
    Rectangle (15,185 181x30), "HP G4 - BH0JPL"
        OnMouseDown: FrameSelectionChange Selection=SelectedFrame=2676ba61-b932-4ea5-9074-f1d3beec8c67, Selection=3, GlobSel=AssignType=Directly, SelType=Locally
    Rectangle (15,290 181x30), "HP G7 - BH0MPL"
        OnMouseDown: FrameSelectionChange Selection=SelectedFrame=2676ba61-b932-4ea5-9074-f1d3beec8c67, Selection=6, GlobSel=AssignType=Directly, SelType=Locally
    Rectangle (15,325 180x55), "Pre Assembly"
    Rectangle (15,385 181x30), "BS02PL.01"
        OnMouseDown: FrameSelectionChange Selection=SelectedFrame=2676ba61-b932-4ea5-9074-f1d3beec8c67, Selection=7, GlobSel=AssignType=Directly, SelType=Locally
    Rectangle (15,150 181x30), "HP G3 - BH0IPL"
        OnMouseDown: FrameSelectionChange Selection=SelectedFrame=2676ba61-b932-4ea5-9074-f1d3beec8c67, Selection=2, GlobSel=AssignType=Directly, SelType=Locally
    Rectangle (15,455 181x30), "BO02PL.01"
        OnMouseDown: FrameSelectionChange Selection=SelectedFrame=2676ba61-b932-4ea5-9074-f1d3beec8c67, Selection=9, GlobSel=AssignType=Directly, SelType=Locally
    Rectangle (15,420 181x30), "BB02PL.01"
        OnMouseDown: FrameSelectionChange Selection=SelectedFrame=2676ba61-b932-4ea5-9074-f1d3beec8c67, Selection=8, GlobSel=AssignType=Directly, SelType=Locally
    Rectangle (15,490 181x30), "BO02PL.02"
        OnMouseDown: FrameSelectionChange Selection=SelectedFrame=2676ba61-b932-4ea5-9074-f1d3beec8c67, Selection=10, GlobSel=AssignType=Directly, SelType=Locally
    Rectangle (15,690 181x30), "BA02PL.03"
        OnMouseDown: FrameSelectionChange Selection=SelectedFrame=2676ba61-b932-4ea5-9074-f1d3beec8c67, Selection=14, GlobSel=AssignType=Directly, SelType=Locally
    Rectangle (15,620 181x30), "BA02PL.01.2"
        OnMouseDown: FrameSelectionChange Selection=SelectedFrame=2676ba61-b932-4ea5-9074-f1d3beec8c67, Selection=12, GlobSel=AssignType=Directly, SelType=Locally
    Rectangle (15,585 181x30), "BA02PL.01.1"
        OnMouseDown: FrameSelectionChange Selection=SelectedFrame=2676ba61-b932-4ea5-9074-f1d3beec8c67, Selection=11, GlobSel=AssignType=Directly, SelType=Locally
    Rectangle (15,655 181x30), "BA02PL.02"
        OnMouseDown: FrameSelectionChange Selection=SelectedFrame=2676ba61-b932-4ea5-9074-f1d3beec8c67, Selection=13, GlobSel=AssignType=Directly, SelType=Locally
    Rectangle (15,220 181x30), "HP G5 - BH0KPL"
        OnMouseDown: FrameSelectionChange Selection=SelectedFrame=2676ba61-b932-4ea5-9074-f1d3beec8c67, Selection=4, GlobSel=AssignType=Directly, SelType=Locally
    Rectangle (15,525 180x55), "Filling Line"
    Rectangle (15,830 181x30), "BA02PL.06.2"
        OnMouseDown: FrameSelectionChange Selection=SelectedFrame=2676ba61-b932-4ea5-9074-f1d3beec8c67, Selection=18, GlobSel=AssignType=Directly, SelType=Locally
    Rectangle (15,760 181x30), "BA02PL.05"
        OnMouseDown: FrameSelectionChange Selection=SelectedFrame=2676ba61-b932-4ea5-9074-f1d3beec8c67, Selection=16, GlobSel=AssignType=Directly, SelType=Locally
    Rectangle (15,725 181x30), "BA02PL.04"
        OnMouseDown: FrameSelectionChange Selection=SelectedFrame=2676ba61-b932-4ea5-9074-f1d3beec8c67, Selection=15, GlobSel=AssignType=Directly, SelType=Locally
    Rectangle (15,795 181x30), "BA02PL.06.1"
        OnMouseDown: FrameSelectionChange Selection=SelectedFrame=2676ba61-b932-4ea5-9074-f1d3beec8c67, Selection=17, GlobSel=AssignType=Directly, SelType=Locally
END_VISUALIZATION

// ---- VISUs/New Visus/vWeighingTunelVisionFrame.TcVIS
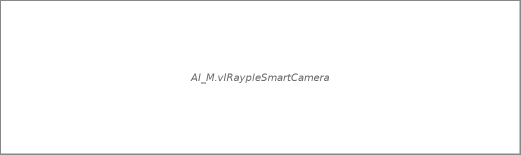
VISUALIZATION vWeighingTunelVisionFrame  // 521x155
    Frame (0,0 521x155)
        shows AI_M.vIRaypleSmartCamera(fb := MAIN.fbSmartCamera)
END_VISUALIZATION

// ---- VISUs/tlNames.TcTLO
TEXTLIST tlNames
  0 = 'Bottle Sensor' | EN: 'Bottle Sensor' | PL: 'Sensor Butelki'
  1 = 'Bottle Eject Sensor' | EN: 'Bottle Eject Sensor' | PL: 'Sensor Wyjazdu Butelki'
  2 = 'Drawer Bottle Sensor' | EN: 'Drawer Bottle Sensor' | PL: 'Sensor Butelki na Szufladzie'
  3 = 'Drawer Lock' | EN: 'Drawer Lock' | PL: 'Zamek Szuflady'
  4 = 'Weight' | EN: 'Weight' | PL: 'Waga'
  5 = 'Out Conveyor' | EN: 'Out Conveyor' | PL: 'Przenosnik Wyjazdowy'
  6 = 'Weighing Actuator' | EN: 'Weighing Actuator' | PL: 'Silownik Wazacy'
  7 = 'Unloading Actuator' | EN: 'Unloading Actuator' | PL: 'Silownik Rozladowujacy'
  8 = 'Pusher Actuator' | EN: 'Pusher Actuator' | PL: 'Silownik Spychajacy'
  9 = 'Separator 1' | EN: 'Separator 1' | PL: 'Separator 1'
  10 = 'Separator 2' | EN: 'Separator 2' | PL: 'Separator 2'
  11 = 'Separator 1 Sensor' | EN: 'Separator 1 Sensor' | PL: 'Separator 1 Czujnik'
  12 = 'Separator 2 Sensor' | EN: 'Separator 2 Sensor' | PL: 'Separator 2 Czujnik'
  13 = 'Table Servo' | EN: 'Table Servo' | PL: 'Table Servo'
   = ''
END_TEXTLIST

// ---- VISUs/tlNamesShort.TcTLO
TEXTLIST tlNamesShort
  0 = 'Bottle Sensor' | EN: 'Bottle Sensor' | PL: 'Sensor Butelki'
  1 = 'Bottle Eject Sensor' | EN: 'Bottle Eject Sensor' | PL: 'Sensor Wyjazdu Butelki'
  2 = 'Drawer Bottle Sensor' | EN: 'Drawer Bottle Sensor' | PL: 'Sensor Butelki na Szufladzie'
  3 = 'Drawer Lock' | EN: 'Drawer Lock' | PL: 'Zamek Szuflady'
  4 = 'Weight' | EN: 'Weight' | PL: 'Waga'
  5 = 'Out Conveyor' | EN: 'Out Conveyor' | PL: 'Przenośnik Wyjazdowy'
  6 = 'Weighing Actuator' | EN: 'Weighing Actuator' | PL: 'Silownik Wazacy'
  7 = 'Unloading Actuator' | EN: 'Unloading Actuator' | PL: 'Silownik Rozladowujacy'
  8 = 'Pusher Actuator' | EN: 'Pusher Actuator' | PL: 'Silownik Spychajacy'
  9 = 'Separator 1' | EN: 'Separator 1' | PL: 'Separator 1'
  10 = 'Separator 2' | EN: 'Separator 2' | PL: 'Separator 2'
  11 = 'Separator 1 Sensor' | EN: 'Separator 1 Sensor' | PL: 'Separator 1 Czujnik'
  12 = 'Separator 2 Sensor' | EN: 'Separator 2 Sensor' | PL: 'Separator 2 Czujnik'
  13 = 'Table Servo' | EN: 'Table Servo' | PL: 'Table Servo'
   = ''
END_TEXTLIST

// ---- VISUs/tlStations.TcTLO
TEXTLIST tlStations
  200 = 'Loading Station' | EN: 'Loading Station' | PL: 'Stacja Ladowania'
  201 = 'Weighing Station' | EN: 'Weighing Station' | PL: 'Stacja Wazenia'
  202 = 'Unloading Station' | EN: 'Unloading Station' | PL: 'Stacja Rozladowania'
   = ''
END_TEXTLIST
